// NeuroPLC — Auto-generated IEC 61131-3 SCL
// Graph: mlp | Target: S71500Backend
// Work memory: 1500KB | LUT points: 50
// Nodes: 8 | Ops: {'matmul': 4, 'standard_act': 2, 'softmax': 1, 'argmax': 1}


DATA_BLOCK "NeuroPLC_Weights"
{ S7_Optimized_Access := 'TRUE' }
VERSION : 0.1
NON_RETAIN

   // MatMul 'fc0': W(32×28) + b(32)
   w0 : Array[0..927] of Real :=
    -0.3770078, 0.3990264, 0.0025516, -0.3593162, 0.1366495, -0.1900285, 0.3891852, -0.1283031,
    -0.3550550, 0.1385999, -0.1855089, -0.3235317, 0.0377216, 0.0437886, -0.2197258, 0.2710523,
    0.4527306, -0.1735796, 0.0918002, -0.2219930, -0.0682289, 0.3726985, -0.4032513, 0.3372299,
    0.1742865, 0.2319893, -0.2549221, -0.3851188, -0.3359332, -0.2109050, 0.2084537, -0.2210156,
    0.2307264, -0.0688108, -0.2107350, -0.1310564, 0.3618010, -0.4616588, 0.1129379, -0.1005827,
    0.2574511, 0.3509765, -0.4043934, 0.0268684, 0.2414633, -0.3012495, -0.1214860, 0.1826331,
    0.1323289, -0.0577001, -0.2709421, -0.1641499, 0.2732217, 0.2441040, -0.0308854, 0.3765655,
    0.4575288, 0.1005922, 0.3384550, 0.3164120, -0.0432535, 0.3674217, 0.2929774, 0.2869964,
    0.4056299, 0.2586457, 0.2159618, -0.0111895, 0.2763612, 0.0318691, -0.2383231, -0.2375112,
    0.1950580, 0.2183585, 0.1430424, 0.1642818, 0.4228715, 0.0093872, -0.1228594, 0.2401115,
    0.3953689, -0.1619427, -0.2964523, 0.2409901, 0.0609418, 0.3946368, 0.4126152, -0.3121379,
    -0.3586196, -0.1127610, 0.1867079, 0.3760083, 0.1564328, 0.1040223, 0.0017305, 0.2251267,
    0.0116038, -0.2901824, -0.0485687, -0.0362714, 0.3139654, 0.1739885, 0.0861147, 0.1815197,
    0.4443266, 0.0452933, 0.2375669, 0.3032796, -0.0065490, 0.0947488, 0.1205690, -0.0489962,
    0.1248455, 0.1040717, -0.1340234, -0.1683266, 0.3904992, 0.0068606, 0.1146591, 0.1519284,
    -0.1746107, -0.2354044, 0.1875906, -0.4197009, -0.4406405, 0.4352002, -0.0388191, -0.0047498,
    -0.1199415, 0.2349747, -0.1049938, -0.1901883, 0.2878532, 0.4529921, 0.1495441, -0.1968838,
    -0.0352187, 0.4251530, 0.1424237, -0.0494499, -0.4578539, 0.4085145, -0.1283757, -0.0146367,
    -0.2926642, -0.3105487, 0.4060314, 0.0523238, -0.0729639, -0.3611083, -0.0152973, -0.2996246,
    -0.1483008, -0.2005807, 0.1901999, 0.2505888, -0.0889782, 0.1222107, 0.2931683, -0.1687088,
    0.3804313, -0.2401819, -0.4427654, -0.1597484, -0.0234017, 0.4053880, 0.1999425, 0.0897930,
    0.2230566, -0.3996429, 0.3089489, -0.1815336, 0.2569048, 0.1170700, 0.4507902, -0.2491009,
    -0.2851968, -0.2911826, 0.1435003, 0.0769116, 0.4312512, 0.1906601, 0.1582011, 0.1911615,
    0.1755516, 0.2151861, 0.1524143, -0.3416874, 0.0968710, 0.2657734, 0.4344491, -0.0455045,
    -0.1944677, 0.0802603, -0.1177095, -0.4598294, -0.3312993, 0.0755498, -0.0593091, 0.0803323,
    0.1532357, 0.2834364, -0.2322901, 0.4257076, 0.0440407, 0.4518892, 0.4534211, -0.2465478,
    -0.2583436, 0.1793744, 0.2255728, -0.1181495, 0.0309696, 0.3416602, 0.1074045, -0.3817922,
    0.2319592, 0.2352205, -0.4058878, -0.2966217, -0.4578832, -0.2983192, 0.1998009, -0.3207857,
    0.1968070, 0.0317941, -0.0459040, 0.4509210, -0.4601454, -0.1890926, -0.3331718, 0.3348714,
    -0.1590407, 0.3725954, -0.3415731, 0.2348770, 0.1108938, -0.1082903, 0.2208081, -0.1398732,
    -0.3844526, -0.3700836, -0.1193436, -0.2816384, 0.2890902, -0.0631509, 0.3378636, -0.3628213,
    0.2885490, 0.4045010, 0.0093051, -0.2111615, 0.3647634, -0.3044274, 0.1587412, -0.1364376,
    0.1600578, -0.1415112, 0.3835287, 0.3839180, 0.3733947, -0.4293965, 0.0489564, 0.3753224,
    -0.4217085, 0.3634868, -0.2955091, -0.0699292, -0.2384017, -0.0102885, -0.3535956, -0.0170217,
    0.1624044, -0.4275157, -0.1322644, -0.2605817, -0.3170779, 0.1670513, 0.4262077, -0.2839059,
    -0.0945041, 0.3597159, -0.3709145, -0.0047849, 0.2313926, -0.1789500, 0.1915937, -0.0686558,
    -0.2433297, 0.2847788, -0.1959274, 0.4444867, -0.3373163, 0.3626398, 0.2917026, 0.2028044,
    0.4221848, -0.4179994, -0.3500787, 0.0961545, -0.2199030, 0.0822042, -0.2083196, 0.0249158,
    -0.4572761, -0.1632026, 0.1749700, -0.0869716, -0.1697042, 0.3751226, 0.1738271, 0.4329614,
    -0.1956948, 0.3490632, -0.3649426, -0.0563313, -0.0793010, -0.4472082, -0.1367153, -0.3672275,
    -0.1686790, 0.1854602, -0.0619579, -0.2322961, 0.1377802, -0.2005911, -0.4102385, 0.1393445,
    0.3889906, -0.1450376, 0.2812740, -0.4401638, -0.3213005, 0.4492195, -0.1869051, 0.2014702,
    0.2808036, 0.0341860, -0.1947227, -0.3475538, -0.0703401, -0.1828323, 0.1945061, 0.2123439,
    0.0289259, -0.4163403, 0.3227376, 0.3735557, 0.4516948, 0.0354091, 0.0885729, 0.3177436,
    -0.0816920, 0.4074438, 0.0901380, -0.2812819, -0.0550214, -0.2856297, 0.0293392, 0.2980039,
    0.4104808, 0.4249691, 0.1168610, 0.0088301, 0.0894373, 0.0541764, -0.3080776, -0.2124508,
    -0.4531886, -0.2822830, 0.4012364, 0.1393107, -0.4608335, -0.3710103, -0.1662148, -0.2561499,
    -0.2994817, -0.3900864, -0.1527744, -0.2041700, 0.4141680, -0.1684453, 0.3008100, -0.0788763,
    -0.1708886, 0.4370478, -0.3517387, -0.2863962, 0.1372241, 0.3990270, -0.0800875, -0.4599121,
    -0.3576341, -0.0551274, -0.1279431, -0.3195898, -0.2090862, 0.3166915, -0.4374981, -0.1036189,
    0.2476588, 0.4534730, 0.0433177, -0.1513664, -0.4313229, 0.3424428, -0.3700289, 0.2864294,
    0.3598893, 0.3942130, 0.4272956, -0.1312214, 0.4043608, -0.1855474, 0.4244733, 0.0673699,
    0.3097988, 0.0743738, -0.0575414, -0.0659323, 0.2604717, 0.2774075, 0.1212956, 0.1247821,
    -0.2054413, -0.4303877, 0.2234309, 0.2691470, 0.2036369, 0.2406268, 0.0806441, -0.0397540,
    0.3085780, 0.3872851, 0.4342453, 0.4615774, -0.0954479, -0.3792063, 0.0337596, 0.1248933,
    -0.3579498, -0.4301034, -0.3439160, 0.2736909, 0.2820499, 0.2041379, 0.3628798, -0.0164372,
    0.4257082, 0.1716245, -0.1405404, -0.1675903, -0.0966237, 0.4509315, -0.2013150, 0.1879556,
    -0.1654160, -0.0369867, -0.1594908, 0.3557843, -0.3484282, 0.0975260, 0.2554502, -0.4486252,
    0.1693635, -0.4568610, -0.0845270, 0.1362543, 0.1075566, -0.4298026, -0.2078513, 0.1131138,
    0.4552583, 0.0955319, -0.0176407, 0.2070304, 0.3496518, 0.0070432, 0.3477424, -0.3328675,
    -0.1949137, -0.4457208, 0.1203264, 0.2554769, -0.4579822, 0.1879786, -0.1129094, 0.2853004,
    0.0644755, -0.3809112, -0.1140574, 0.4154554, 0.1054994, 0.4068863, -0.2891253, 0.0136368,
    -0.0689342, -0.4286978, 0.2200271, 0.0348938, -0.3910995, 0.4048684, -0.4127417, -0.2598001,
    0.2112517, -0.1751920, -0.4369283, -0.1871661, 0.0023222, 0.4015321, 0.2616409, -0.3857000,
    -0.2690184, 0.3857079, -0.2387726, 0.2434377, 0.0714437, 0.0578954, -0.2566555, 0.2605321,
    0.0101752, 0.1413683, 0.0509943, -0.3524976, 0.1041765, 0.4223077, 0.3136883, 0.1300556,
    0.4291077, 0.2816193, 0.1022774, -0.3548588, 0.0421972, -0.2862138, -0.0118091, -0.4334079,
    -0.1866055, 0.0868014, 0.1372423, -0.1925206, 0.0754342, -0.1125624, 0.4365539, 0.2470605,
    0.4543210, -0.2610196, 0.2990730, -0.3651120, 0.1277550, 0.2837237, -0.0998289, 0.0588385,
    0.3020812, 0.3680393, -0.3858286, 0.0961783, 0.4596364, -0.2120740, -0.4344158, -0.3728840,
    0.1881307, -0.1419628, -0.2620887, -0.1069769, 0.1167762, 0.0211368, 0.1347501, -0.3661770,
    0.0150048, -0.3614159, 0.2448329, 0.2522876, 0.1993004, -0.0491755, -0.3745691, -0.2868368,
    -0.3422473, 0.2306486, -0.0107990, -0.2471329, 0.4094761, 0.4462330, -0.1006898, -0.3417571,
    -0.3526864, 0.3459129, -0.1873048, -0.3418673, 0.1899261, -0.4220347, 0.4099078, -0.0792820,
    0.4320456, -0.1785485, 0.3833564, -0.1475922, 0.2927010, -0.3002279, 0.4024807, -0.2212537,
    0.1185881, 0.0967595, -0.2608397, -0.0318049, -0.0925073, -0.0683086, -0.4334753, -0.3877276,
    0.2818044, 0.3985909, 0.1276854, 0.1431718, 0.0759905, 0.2359956, -0.3075322, -0.4488399,
    0.3382713, 0.0587753, 0.1603718, 0.2061060, 0.4003389, 0.0745798, -0.1383399, 0.0690251,
    -0.3627133, -0.2600157, 0.2113945, -0.0398504, 0.3121908, -0.0397190, -0.2176074, 0.2885886,
    0.2448370, 0.2249159, 0.3732608, 0.1413454, 0.2938702, 0.0381091, -0.0704973, -0.0676246,
    -0.3967757, 0.1924810, 0.0945449, -0.2569663, 0.0901330, -0.1480842, -0.1106209, -0.0419426,
    0.1201892, -0.3996566, 0.1597114, 0.1156000, -0.3738315, -0.0122839, 0.0922182, 0.1364632,
    -0.0856640, 0.3560283, 0.4043280, -0.2908444, 0.1349952, -0.4130700, -0.4436539, -0.1325469,
    -0.1949083, -0.0976171, 0.1365751, -0.2287472, 0.2230470, -0.2904527, -0.1090742, 0.2397174,
    0.2679743, 0.4155956, 0.4056778, -0.2658896, -0.2220807, -0.4523228, 0.0380185, 0.2802896,
    -0.3090282, -0.0251335, 0.2784542, -0.1911104, 0.1081119, -0.1071131, -0.2883627, 0.1024943,
    0.1079664, 0.0528435, 0.0637380, 0.1360845, 0.2319627, -0.4568143, 0.1126708, 0.2881851,
    -0.0390266, -0.3154065, -0.1891240, 0.3152807, -0.3991016, -0.1147000, -0.1755120, -0.0517076,
    0.2942899, -0.1193079, 0.3693818, 0.3813385, -0.3667921, 0.3955849, -0.3730764, 0.2449901,
    0.4367092, -0.4306898, -0.0932055, -0.2762457, 0.0764579, -0.0612213, 0.3295913, 0.1819134,
    0.3777595, -0.2319842, -0.2136903, -0.0318793, -0.3945642, 0.4148945, 0.1171657, 0.1796898,
    -0.3446222, -0.2104773, 0.0936033, -0.2603089, -0.2805420, -0.4435062, 0.3793530, 0.0610302,
    0.2015716, -0.3638270, 0.0155152, -0.2831283, -0.4584919, 0.3411648, -0.0253624, 0.0896016,
    -0.3085061, 0.3751078, 0.3812718, -0.2918622, 0.2093002, -0.3870984, -0.4346099, 0.3052061,
    0.2963735, -0.4020928, -0.1916119, 0.4596418, -0.2036503, -0.1675266, -0.3643405, -0.0234888,
    0.1632566, 0.2617638, -0.0987748, 0.2144748, 0.3578448, 0.4327554, -0.2301966, -0.1355437,
    0.3251480, -0.0650652, 0.4607093, 0.4538801, 0.3257216, 0.2937019, 0.2583465, 0.0784602,
    -0.2065715, 0.2250659, 0.4356502, -0.0072217, -0.1376927, 0.0364345, -0.3187408, 0.3734230,
    -0.2510726, -0.1775467, -0.3211187, -0.3278403, -0.3991595, 0.0120480, 0.4284748, 0.1523868,
    0.2492753, -0.4192764, -0.4125061, -0.1992944, -0.3151319, -0.4228379, 0.2395529, -0.3589366,
    -0.4471393, 0.1070668, 0.0736012, -0.1881842, 0.1677683, -0.2855140, 0.0012233, -0.4301678,
    0.4539815, -0.2786066, -0.4277930, 0.1925392, -0.4242253, 0.0287630, 0.3206151, 0.4489035,
    -0.3228373, 0.0110811, 0.1304550, 0.3193927, -0.1024946, -0.3389935, -0.0040539, -0.3283602,
    0.3610852, 0.3990757, 0.3903281, 0.2358855, 0.3887415, -0.4240198, 0.1866908, -0.4352202,
    0.4117475, -0.3510597, -0.3075358, -0.4001069, -0.3420205, 0.3339028, -0.1180067, -0.0772094,
    0.2149267, -0.3405320, -0.2175644, 0.2114443, -0.0852025, -0.1429342, -0.4322555, -0.0152842,
    -0.3777024, 0.3303320, 0.0268890, 0.0038649, 0.2427567, -0.1545651, -0.0877347, 0.1801398,
    -0.0444975, 0.2461711, -0.4585460, -0.4603382, 0.3602494, -0.3180314, 0.4038997, 0.3527558,
    0.0713230, -0.0322537, -0.0798554, -0.3169685, 0.2551405, -0.1615019, 0.1647311, 0.4458464,
    0.2310456, -0.0397924, -0.0218926, -0.2396226, -0.2713118, -0.1628663, 0.1717695, 0.1115326,
    -0.1871466, -0.2292732, 0.0375844, 0.2459664, 0.4030566, -0.3787265, 0.2261490, 0.2506774,
    0.0796954, -0.3811616, -0.4266883, -0.4610847, -0.2181492, 0.0805867, -0.1990638, -0.3294418,
    0.0, 0.0, 0.0, 0.0, 0.0, 0.0, 0.0, 0.0,
    0.0, 0.0, 0.0, 0.0, 0.0, 0.0, 0.0, 0.0,
    0.0, 0.0, 0.0, 0.0, 0.0, 0.0, 0.0, 0.0,
    0.0, 0.0, 0.0, 0.0, 0.0, 0.0, 0.0, 0.0;

   // MatMul 'fc1': W(16×32) + b(16)
   w1 : Array[0..527] of Real :=
    -0.3935522, -0.1891568, -0.2444881, -0.2520988, 0.0168740, -0.0661420, -0.0739836, 0.1249234,
    0.0495841, -0.3324362, 0.3990199, -0.3827971, 0.1509344, 0.2727351, 0.1899064, 0.1232548,
    -0.1740977, 0.3996815, -0.0156190, 0.4319531, 0.2304519, 0.2019619, -0.1108288, 0.2639450,
    -0.3004889, 0.2053759, -0.2507130, -0.1099108, 0.3508554, 0.2798605, 0.3080718, -0.2521698,
    0.0398361, 0.0467716, 0.3878656, -0.0975975, 0.2259126, -0.2130022, 0.2817706, -0.4208167,
    0.2917084, 0.4064464, 0.1718341, 0.1449949, -0.2451592, 0.2201938, -0.1602577, -0.3822802,
    -0.1150226, -0.2497750, -0.4201412, -0.0156258, -0.1511233, -0.3021594, -0.1100701, 0.3851436,
    -0.2900417, 0.1651725, 0.2725570, -0.2857571, -0.1159424, 0.3958912, -0.4076339, 0.2155754,
    -0.3153985, 0.1522842, 0.2238676, 0.0359937, -0.2988871, -0.1637969, 0.2320338, 0.0857368,
    0.1976208, 0.0608633, -0.1173251, -0.3213641, -0.0849160, 0.1718496, 0.1879434, 0.3173548,
    0.1776288, -0.2859888, 0.4273638, -0.0753660, 0.2396645, -0.1966574, 0.3941564, -0.4111311,
    0.4031409, 0.3382389, 0.2827366, 0.3812202, -0.4018011, 0.2268997, -0.4327545, 0.0562466,
    -0.4181275, 0.0895361, 0.0215759, -0.4292598, -0.0456185, 0.3361736, 0.1588783, -0.3002315,
    0.1648912, 0.2550659, 0.1932670, 0.3281942, 0.2067506, -0.4133190, -0.1431655, 0.4150747,
    0.3473578, 0.3837779, 0.0933603, 0.2324348, 0.2446682, -0.2923857, -0.1816045, 0.0872757,
    -0.1632624, 0.0132405, 0.0319080, -0.3656984, -0.0171522, 0.4021245, -0.4298175, -0.1553442,
    -0.0378739, -0.0558841, -0.1237145, 0.2343058, -0.3540494, 0.0363749, -0.1224368, 0.1096888,
    0.1723547, 0.2546408, 0.3474467, -0.2087996, 0.4150974, 0.2533172, -0.3616572, -0.1398576,
    0.1326821, 0.0146453, 0.3335588, 0.1515740, -0.1683524, -0.0804338, 0.4306846, 0.0640880,
    0.2288128, 0.0326079, 0.1973397, 0.0868359, 0.3189215, 0.1261115, 0.4030693, 0.0196063,
    0.1143374, -0.1861071, -0.3970583, 0.4306547, 0.3728819, -0.1188974, -0.2829262, -0.3271297,
    -0.2453017, 0.1782900, -0.0166697, -0.3631355, -0.1097839, 0.0609611, 0.0001612, 0.3813087,
    0.1942296, -0.3436415, -0.3196552, -0.3243870, 0.2198140, 0.3918344, 0.0912264, 0.2238992,
    -0.3022591, 0.3621037, 0.3434459, -0.1731028, 0.3113935, 0.3348374, 0.2629885, 0.0019000,
    0.3024160, -0.0626668, -0.0818046, -0.3892852, -0.1082816, -0.2291101, 0.1406163, -0.3290255,
    0.0634920, -0.0686606, 0.1352782, -0.2557390, 0.3506733, -0.2629621, -0.2691220, -0.2397180,
    -0.2910091, 0.0893200, 0.1797454, 0.2301134, -0.3933525, 0.0697611, -0.1224633, -0.1336698,
    0.0822801, 0.0491940, 0.1768592, -0.1431975, 0.1519364, 0.2522070, -0.3521394, -0.3634867,
    0.3611591, 0.0925913, 0.3470873, 0.0306298, 0.3107211, -0.1883461, 0.2165535, -0.1091567,
    0.0689959, 0.3486420, -0.1837859, 0.0694401, 0.2055986, 0.2386295, 0.3321949, 0.1919344,
    0.4253771, -0.3774826, -0.0617012, 0.0334252, 0.3778329, 0.2201037, -0.2276398, 0.1301410,
    0.3501653, 0.2798014, 0.4256953, -0.1441793, -0.0663480, -0.4205136, 0.3892752, -0.3286948,
    0.0955538, 0.3663456, -0.1591998, 0.3128131, 0.0344288, 0.0733947, -0.2083270, -0.3181835,
    0.2916943, 0.1976334, -0.0215316, -0.1335652, -0.1110399, -0.4227563, -0.2664171, 0.4199895,
    -0.3832088, 0.0912991, 0.3962664, -0.2253252, -0.4168374, -0.0803243, -0.2418978, 0.2176948,
    -0.3986563, -0.0865313, -0.1186279, -0.4000811, 0.0561389, -0.1613197, -0.4163839, 0.1215905,
    -0.1568890, 0.3878794, 0.3653413, -0.2158771, -0.0794441, 0.0936781, 0.2255915, 0.3624552,
    0.2718166, -0.0088999, -0.2009125, 0.0077918, 0.1461028, 0.2432971, 0.1760126, 0.1427329,
    -0.0146298, -0.3526535, -0.1145816, 0.0303672, -0.3133373, 0.3928600, 0.3592887, 0.3393191,
    0.2999697, -0.2127717, -0.3682398, -0.2014481, 0.2898328, -0.0393004, 0.3296660, -0.2576033,
    -0.2580386, 0.3286115, 0.3484521, 0.1741413, -0.3222574, 0.4139940, -0.2123599, -0.0532465,
    -0.1246679, -0.1157071, -0.3183327, 0.0137842, 0.1334311, -0.0707376, -0.1285511, -0.4081723,
    -0.1506712, 0.2322767, 0.0759037, 0.3221440, 0.2789797, -0.3218980, -0.0615748, -0.3991559,
    -0.4185835, -0.2636460, -0.1289205, 0.2750368, 0.2876762, -0.3447819, -0.1141558, 0.1948618,
    -0.1709883, 0.3542524, -0.1556085, -0.0569944, 0.2803813, 0.0518793, -0.0245967, 0.1485651,
    -0.0932260, 0.2044456, -0.3843631, 0.1491727, -0.1015462, 0.0335794, -0.2548426, -0.2155586,
    0.3438183, -0.3987876, -0.1833805, -0.3147031, -0.4217897, 0.4175099, -0.0144855, -0.3033746,
    -0.1601701, 0.3044005, -0.0549371, -0.2065555, -0.2234019, -0.3457984, -0.0095058, 0.4049891,
    0.1624429, -0.0648286, 0.3860819, 0.1274094, 0.2339818, 0.1994726, -0.3863117, -0.3547160,
    0.2731713, 0.3852477, -0.0738010, 0.4109565, 0.3464701, 0.2911135, -0.2596304, -0.3724965,
    -0.0749315, -0.0193869, -0.2211102, -0.2740593, -0.3613006, 0.2223929, -0.0702648, 0.1260325,
    -0.3447631, 0.2582121, 0.1769404, 0.4101386, -0.2221670, 0.4048361, -0.2569288, 0.1401117,
    -0.3058916, 0.2899141, -0.2516046, -0.0204311, 0.3705838, 0.4224865, -0.0464628, 0.2932765,
    -0.1048749, -0.1260871, 0.1966383, 0.3772893, 0.0665107, 0.4117973, 0.3348016, -0.3298126,
    0.1286661, -0.3882708, 0.0985853, 0.2120279, 0.2686936, -0.2604558, -0.1903019, 0.1670984,
    0.1759086, -0.2155941, -0.4271439, -0.1347190, 0.3518137, 0.1066233, -0.0060884, -0.0989732,
    -0.1571809, 0.2292162, -0.2883213, 0.1154139, 0.2343982, -0.0461321, -0.2751803, -0.0112296,
    0.2915563, 0.3558245, 0.2112975, -0.2306676, -0.3320167, 0.2315517, -0.0035513, 0.3149335,
    0.0999751, -0.0704947, -0.3919639, -0.0087440, -0.1189045, -0.3321721, 0.0222524, -0.3617505,
    -0.1745312, 0.0928437, 0.3209649, 0.4192130, 0.0815147, 0.2839914, 0.0094900, 0.3304590,
    0.1507888, -0.1633613, -0.2137657, 0.4228123, -0.0633699, -0.3235189, -0.3633914, 0.0783406,
    0.2527627, 0.4272875, -0.2854069, 0.1855697, -0.1320681, 0.3007466, 0.0956593, -0.2299400,
    0.0410553, 0.0255588, -0.2430910, 0.1599361, 0.2384051, 0.0154256, 0.2833597, 0.0843526,
    0.3284023, 0.1945453, 0.1661874, 0.1049307, -0.3034132, 0.1947828, 0.3134930, -0.1473352,
    0.0, 0.0, 0.0, 0.0, 0.0, 0.0, 0.0, 0.0,
    0.0, 0.0, 0.0, 0.0, 0.0, 0.0, 0.0, 0.0;

   // MatMul 'fc2': W(4×16) + b(4)
   w2 : Array[0..67] of Real :=
    0.3119249, -0.6119898, 0.2570214, -0.5775461, -0.3303460, -0.0226893, -0.0253589, 0.0133041,
    0.2119226, 0.1795658, 0.1164464, -0.5784835, 0.4102349, -0.5724207, -0.5247188, 0.2892720,
    0.0710802, 0.4088987, -0.4011595, 0.1927266, 0.0227786, -0.3939466, 0.5633335, 0.4811944,
    0.4671021, -0.4038831, 0.2076768, -0.5081061, 0.1620483, -0.2713509, 0.4681324, 0.3022301,
    0.3770372, -0.5370517, -0.1928490, 0.0872999, -0.0823838, -0.2322832, 0.0953737, -0.0633100,
    -0.2465645, 0.4775037, 0.5268021, -0.1162953, -0.3230001, 0.2317193, 0.2054757, -0.4918106,
    0.2500432, -0.1568022, -0.4481698, 0.3745956, -0.0458250, -0.5208440, 0.1315344, 0.3012816,
    0.4046838, -0.6074986, 0.0947582, -0.3567927, 0.0561409, 0.1993957, 0.1098667, 0.0024996,
    0.0, 0.0, 0.0, 0.0;

   // Total: 3 array blocks
END_DATA_BLOCK

FUNCTION_BLOCK "NeuroPLC_Inference"
{ S7_Optimized_Access := 'TRUE' }
VERSION : 0.1
VAR_INPUT
    features : Array[0..27] of Real;
END_VAR

VAR_OUTPUT
    fault_class : Int;
    confidence : Real;
END_VAR

VAR
    i, j, k : Int;
    sum_val, max_val, t_val : Real;
    v0 : Array[0..27] of Real;
    v1 : Array[0..31] of Real;
    v2 : Array[0..31] of Real;
    v3 : Array[0..15] of Real;
    v4 : Array[0..15] of Real;
    v5 : Array[0..3] of Real;
    v6 : Array[0..3] of Real;
END_VAR

BEGIN
    // ---- Input ----
    FOR i := 0 TO 27 DO
        v0[i] := features[i];
    END_FOR;

    // ---- fc0: MatMul(28→32) ----
    // W = "NeuroPLC_Weights".w0[:896],   b = w0[896:]
    v1[0] := "NeuroPLC_Weights".w0[896 + 0] + "NeuroPLC_Weights".w0[0] * v0[0] + "NeuroPLC_Weights".w0[1] * v0[1] + "NeuroPLC_Weights".w0[2] * v0[2] + "NeuroPLC_Weights".w0[3] * v0[3] + "NeuroPLC_Weights".w0[4] * v0[4] + "NeuroPLC_Weights".w0[5] * v0[5] + "NeuroPLC_Weights".w0[6] * v0[6] + "NeuroPLC_Weights".w0[7] * v0[7] + "NeuroPLC_Weights".w0[8] * v0[8] + "NeuroPLC_Weights".w0[9] * v0[9] + "NeuroPLC_Weights".w0[10] * v0[10] + "NeuroPLC_Weights".w0[11] * v0[11] + "NeuroPLC_Weights".w0[12] * v0[12] + "NeuroPLC_Weights".w0[13] * v0[13] + "NeuroPLC_Weights".w0[14] * v0[14] + "NeuroPLC_Weights".w0[15] * v0[15] + "NeuroPLC_Weights".w0[16] * v0[16] + "NeuroPLC_Weights".w0[17] * v0[17] + "NeuroPLC_Weights".w0[18] * v0[18] + "NeuroPLC_Weights".w0[19] * v0[19] + "NeuroPLC_Weights".w0[20] * v0[20] + "NeuroPLC_Weights".w0[21] * v0[21] + "NeuroPLC_Weights".w0[22] * v0[22] + "NeuroPLC_Weights".w0[23] * v0[23] + "NeuroPLC_Weights".w0[24] * v0[24] + "NeuroPLC_Weights".w0[25] * v0[25] + "NeuroPLC_Weights".w0[26] * v0[26] + "NeuroPLC_Weights".w0[27] * v0[27];
    v1[1] := "NeuroPLC_Weights".w0[896 + 1] + "NeuroPLC_Weights".w0[28] * v0[0] + "NeuroPLC_Weights".w0[29] * v0[1] + "NeuroPLC_Weights".w0[30] * v0[2] + "NeuroPLC_Weights".w0[31] * v0[3] + "NeuroPLC_Weights".w0[32] * v0[4] + "NeuroPLC_Weights".w0[33] * v0[5] + "NeuroPLC_Weights".w0[34] * v0[6] + "NeuroPLC_Weights".w0[35] * v0[7] + "NeuroPLC_Weights".w0[36] * v0[8] + "NeuroPLC_Weights".w0[37] * v0[9] + "NeuroPLC_Weights".w0[38] * v0[10] + "NeuroPLC_Weights".w0[39] * v0[11] + "NeuroPLC_Weights".w0[40] * v0[12] + "NeuroPLC_Weights".w0[41] * v0[13] + "NeuroPLC_Weights".w0[42] * v0[14] + "NeuroPLC_Weights".w0[43] * v0[15] + "NeuroPLC_Weights".w0[44] * v0[16] + "NeuroPLC_Weights".w0[45] * v0[17] + "NeuroPLC_Weights".w0[46] * v0[18] + "NeuroPLC_Weights".w0[47] * v0[19] + "NeuroPLC_Weights".w0[48] * v0[20] + "NeuroPLC_Weights".w0[49] * v0[21] + "NeuroPLC_Weights".w0[50] * v0[22] + "NeuroPLC_Weights".w0[51] * v0[23] + "NeuroPLC_Weights".w0[52] * v0[24] + "NeuroPLC_Weights".w0[53] * v0[25] + "NeuroPLC_Weights".w0[54] * v0[26] + "NeuroPLC_Weights".w0[55] * v0[27];
    v1[2] := "NeuroPLC_Weights".w0[896 + 2] + "NeuroPLC_Weights".w0[56] * v0[0] + "NeuroPLC_Weights".w0[57] * v0[1] + "NeuroPLC_Weights".w0[58] * v0[2] + "NeuroPLC_Weights".w0[59] * v0[3] + "NeuroPLC_Weights".w0[60] * v0[4] + "NeuroPLC_Weights".w0[61] * v0[5] + "NeuroPLC_Weights".w0[62] * v0[6] + "NeuroPLC_Weights".w0[63] * v0[7] + "NeuroPLC_Weights".w0[64] * v0[8] + "NeuroPLC_Weights".w0[65] * v0[9] + "NeuroPLC_Weights".w0[66] * v0[10] + "NeuroPLC_Weights".w0[67] * v0[11] + "NeuroPLC_Weights".w0[68] * v0[12] + "NeuroPLC_Weights".w0[69] * v0[13] + "NeuroPLC_Weights".w0[70] * v0[14] + "NeuroPLC_Weights".w0[71] * v0[15] + "NeuroPLC_Weights".w0[72] * v0[16] + "NeuroPLC_Weights".w0[73] * v0[17] + "NeuroPLC_Weights".w0[74] * v0[18] + "NeuroPLC_Weights".w0[75] * v0[19] + "NeuroPLC_Weights".w0[76] * v0[20] + "NeuroPLC_Weights".w0[77] * v0[21] + "NeuroPLC_Weights".w0[78] * v0[22] + "NeuroPLC_Weights".w0[79] * v0[23] + "NeuroPLC_Weights".w0[80] * v0[24] + "NeuroPLC_Weights".w0[81] * v0[25] + "NeuroPLC_Weights".w0[82] * v0[26] + "NeuroPLC_Weights".w0[83] * v0[27];
    v1[3] := "NeuroPLC_Weights".w0[896 + 3] + "NeuroPLC_Weights".w0[84] * v0[0] + "NeuroPLC_Weights".w0[85] * v0[1] + "NeuroPLC_Weights".w0[86] * v0[2] + "NeuroPLC_Weights".w0[87] * v0[3] + "NeuroPLC_Weights".w0[88] * v0[4] + "NeuroPLC_Weights".w0[89] * v0[5] + "NeuroPLC_Weights".w0[90] * v0[6] + "NeuroPLC_Weights".w0[91] * v0[7] + "NeuroPLC_Weights".w0[92] * v0[8] + "NeuroPLC_Weights".w0[93] * v0[9] + "NeuroPLC_Weights".w0[94] * v0[10] + "NeuroPLC_Weights".w0[95] * v0[11] + "NeuroPLC_Weights".w0[96] * v0[12] + "NeuroPLC_Weights".w0[97] * v0[13] + "NeuroPLC_Weights".w0[98] * v0[14] + "NeuroPLC_Weights".w0[99] * v0[15] + "NeuroPLC_Weights".w0[100] * v0[16] + "NeuroPLC_Weights".w0[101] * v0[17] + "NeuroPLC_Weights".w0[102] * v0[18] + "NeuroPLC_Weights".w0[103] * v0[19] + "NeuroPLC_Weights".w0[104] * v0[20] + "NeuroPLC_Weights".w0[105] * v0[21] + "NeuroPLC_Weights".w0[106] * v0[22] + "NeuroPLC_Weights".w0[107] * v0[23] + "NeuroPLC_Weights".w0[108] * v0[24] + "NeuroPLC_Weights".w0[109] * v0[25] + "NeuroPLC_Weights".w0[110] * v0[26] + "NeuroPLC_Weights".w0[111] * v0[27];
    v1[4] := "NeuroPLC_Weights".w0[896 + 4] + "NeuroPLC_Weights".w0[112] * v0[0] + "NeuroPLC_Weights".w0[113] * v0[1] + "NeuroPLC_Weights".w0[114] * v0[2] + "NeuroPLC_Weights".w0[115] * v0[3] + "NeuroPLC_Weights".w0[116] * v0[4] + "NeuroPLC_Weights".w0[117] * v0[5] + "NeuroPLC_Weights".w0[118] * v0[6] + "NeuroPLC_Weights".w0[119] * v0[7] + "NeuroPLC_Weights".w0[120] * v0[8] + "NeuroPLC_Weights".w0[121] * v0[9] + "NeuroPLC_Weights".w0[122] * v0[10] + "NeuroPLC_Weights".w0[123] * v0[11] + "NeuroPLC_Weights".w0[124] * v0[12] + "NeuroPLC_Weights".w0[125] * v0[13] + "NeuroPLC_Weights".w0[126] * v0[14] + "NeuroPLC_Weights".w0[127] * v0[15] + "NeuroPLC_Weights".w0[128] * v0[16] + "NeuroPLC_Weights".w0[129] * v0[17] + "NeuroPLC_Weights".w0[130] * v0[18] + "NeuroPLC_Weights".w0[131] * v0[19] + "NeuroPLC_Weights".w0[132] * v0[20] + "NeuroPLC_Weights".w0[133] * v0[21] + "NeuroPLC_Weights".w0[134] * v0[22] + "NeuroPLC_Weights".w0[135] * v0[23] + "NeuroPLC_Weights".w0[136] * v0[24] + "NeuroPLC_Weights".w0[137] * v0[25] + "NeuroPLC_Weights".w0[138] * v0[26] + "NeuroPLC_Weights".w0[139] * v0[27];
    v1[5] := "NeuroPLC_Weights".w0[896 + 5] + "NeuroPLC_Weights".w0[140] * v0[0] + "NeuroPLC_Weights".w0[141] * v0[1] + "NeuroPLC_Weights".w0[142] * v0[2] + "NeuroPLC_Weights".w0[143] * v0[3] + "NeuroPLC_Weights".w0[144] * v0[4] + "NeuroPLC_Weights".w0[145] * v0[5] + "NeuroPLC_Weights".w0[146] * v0[6] + "NeuroPLC_Weights".w0[147] * v0[7] + "NeuroPLC_Weights".w0[148] * v0[8] + "NeuroPLC_Weights".w0[149] * v0[9] + "NeuroPLC_Weights".w0[150] * v0[10] + "NeuroPLC_Weights".w0[151] * v0[11] + "NeuroPLC_Weights".w0[152] * v0[12] + "NeuroPLC_Weights".w0[153] * v0[13] + "NeuroPLC_Weights".w0[154] * v0[14] + "NeuroPLC_Weights".w0[155] * v0[15] + "NeuroPLC_Weights".w0[156] * v0[16] + "NeuroPLC_Weights".w0[157] * v0[17] + "NeuroPLC_Weights".w0[158] * v0[18] + "NeuroPLC_Weights".w0[159] * v0[19] + "NeuroPLC_Weights".w0[160] * v0[20] + "NeuroPLC_Weights".w0[161] * v0[21] + "NeuroPLC_Weights".w0[162] * v0[22] + "NeuroPLC_Weights".w0[163] * v0[23] + "NeuroPLC_Weights".w0[164] * v0[24] + "NeuroPLC_Weights".w0[165] * v0[25] + "NeuroPLC_Weights".w0[166] * v0[26] + "NeuroPLC_Weights".w0[167] * v0[27];
    v1[6] := "NeuroPLC_Weights".w0[896 + 6] + "NeuroPLC_Weights".w0[168] * v0[0] + "NeuroPLC_Weights".w0[169] * v0[1] + "NeuroPLC_Weights".w0[170] * v0[2] + "NeuroPLC_Weights".w0[171] * v0[3] + "NeuroPLC_Weights".w0[172] * v0[4] + "NeuroPLC_Weights".w0[173] * v0[5] + "NeuroPLC_Weights".w0[174] * v0[6] + "NeuroPLC_Weights".w0[175] * v0[7] + "NeuroPLC_Weights".w0[176] * v0[8] + "NeuroPLC_Weights".w0[177] * v0[9] + "NeuroPLC_Weights".w0[178] * v0[10] + "NeuroPLC_Weights".w0[179] * v0[11] + "NeuroPLC_Weights".w0[180] * v0[12] + "NeuroPLC_Weights".w0[181] * v0[13] + "NeuroPLC_Weights".w0[182] * v0[14] + "NeuroPLC_Weights".w0[183] * v0[15] + "NeuroPLC_Weights".w0[184] * v0[16] + "NeuroPLC_Weights".w0[185] * v0[17] + "NeuroPLC_Weights".w0[186] * v0[18] + "NeuroPLC_Weights".w0[187] * v0[19] + "NeuroPLC_Weights".w0[188] * v0[20] + "NeuroPLC_Weights".w0[189] * v0[21] + "NeuroPLC_Weights".w0[190] * v0[22] + "NeuroPLC_Weights".w0[191] * v0[23] + "NeuroPLC_Weights".w0[192] * v0[24] + "NeuroPLC_Weights".w0[193] * v0[25] + "NeuroPLC_Weights".w0[194] * v0[26] + "NeuroPLC_Weights".w0[195] * v0[27];
    v1[7] := "NeuroPLC_Weights".w0[896 + 7] + "NeuroPLC_Weights".w0[196] * v0[0] + "NeuroPLC_Weights".w0[197] * v0[1] + "NeuroPLC_Weights".w0[198] * v0[2] + "NeuroPLC_Weights".w0[199] * v0[3] + "NeuroPLC_Weights".w0[200] * v0[4] + "NeuroPLC_Weights".w0[201] * v0[5] + "NeuroPLC_Weights".w0[202] * v0[6] + "NeuroPLC_Weights".w0[203] * v0[7] + "NeuroPLC_Weights".w0[204] * v0[8] + "NeuroPLC_Weights".w0[205] * v0[9] + "NeuroPLC_Weights".w0[206] * v0[10] + "NeuroPLC_Weights".w0[207] * v0[11] + "NeuroPLC_Weights".w0[208] * v0[12] + "NeuroPLC_Weights".w0[209] * v0[13] + "NeuroPLC_Weights".w0[210] * v0[14] + "NeuroPLC_Weights".w0[211] * v0[15] + "NeuroPLC_Weights".w0[212] * v0[16] + "NeuroPLC_Weights".w0[213] * v0[17] + "NeuroPLC_Weights".w0[214] * v0[18] + "NeuroPLC_Weights".w0[215] * v0[19] + "NeuroPLC_Weights".w0[216] * v0[20] + "NeuroPLC_Weights".w0[217] * v0[21] + "NeuroPLC_Weights".w0[218] * v0[22] + "NeuroPLC_Weights".w0[219] * v0[23] + "NeuroPLC_Weights".w0[220] * v0[24] + "NeuroPLC_Weights".w0[221] * v0[25] + "NeuroPLC_Weights".w0[222] * v0[26] + "NeuroPLC_Weights".w0[223] * v0[27];
    v1[8] := "NeuroPLC_Weights".w0[896 + 8] + "NeuroPLC_Weights".w0[224] * v0[0] + "NeuroPLC_Weights".w0[225] * v0[1] + "NeuroPLC_Weights".w0[226] * v0[2] + "NeuroPLC_Weights".w0[227] * v0[3] + "NeuroPLC_Weights".w0[228] * v0[4] + "NeuroPLC_Weights".w0[229] * v0[5] + "NeuroPLC_Weights".w0[230] * v0[6] + "NeuroPLC_Weights".w0[231] * v0[7] + "NeuroPLC_Weights".w0[232] * v0[8] + "NeuroPLC_Weights".w0[233] * v0[9] + "NeuroPLC_Weights".w0[234] * v0[10] + "NeuroPLC_Weights".w0[235] * v0[11] + "NeuroPLC_Weights".w0[236] * v0[12] + "NeuroPLC_Weights".w0[237] * v0[13] + "NeuroPLC_Weights".w0[238] * v0[14] + "NeuroPLC_Weights".w0[239] * v0[15] + "NeuroPLC_Weights".w0[240] * v0[16] + "NeuroPLC_Weights".w0[241] * v0[17] + "NeuroPLC_Weights".w0[242] * v0[18] + "NeuroPLC_Weights".w0[243] * v0[19] + "NeuroPLC_Weights".w0[244] * v0[20] + "NeuroPLC_Weights".w0[245] * v0[21] + "NeuroPLC_Weights".w0[246] * v0[22] + "NeuroPLC_Weights".w0[247] * v0[23] + "NeuroPLC_Weights".w0[248] * v0[24] + "NeuroPLC_Weights".w0[249] * v0[25] + "NeuroPLC_Weights".w0[250] * v0[26] + "NeuroPLC_Weights".w0[251] * v0[27];
    v1[9] := "NeuroPLC_Weights".w0[896 + 9] + "NeuroPLC_Weights".w0[252] * v0[0] + "NeuroPLC_Weights".w0[253] * v0[1] + "NeuroPLC_Weights".w0[254] * v0[2] + "NeuroPLC_Weights".w0[255] * v0[3] + "NeuroPLC_Weights".w0[256] * v0[4] + "NeuroPLC_Weights".w0[257] * v0[5] + "NeuroPLC_Weights".w0[258] * v0[6] + "NeuroPLC_Weights".w0[259] * v0[7] + "NeuroPLC_Weights".w0[260] * v0[8] + "NeuroPLC_Weights".w0[261] * v0[9] + "NeuroPLC_Weights".w0[262] * v0[10] + "NeuroPLC_Weights".w0[263] * v0[11] + "NeuroPLC_Weights".w0[264] * v0[12] + "NeuroPLC_Weights".w0[265] * v0[13] + "NeuroPLC_Weights".w0[266] * v0[14] + "NeuroPLC_Weights".w0[267] * v0[15] + "NeuroPLC_Weights".w0[268] * v0[16] + "NeuroPLC_Weights".w0[269] * v0[17] + "NeuroPLC_Weights".w0[270] * v0[18] + "NeuroPLC_Weights".w0[271] * v0[19] + "NeuroPLC_Weights".w0[272] * v0[20] + "NeuroPLC_Weights".w0[273] * v0[21] + "NeuroPLC_Weights".w0[274] * v0[22] + "NeuroPLC_Weights".w0[275] * v0[23] + "NeuroPLC_Weights".w0[276] * v0[24] + "NeuroPLC_Weights".w0[277] * v0[25] + "NeuroPLC_Weights".w0[278] * v0[26] + "NeuroPLC_Weights".w0[279] * v0[27];
    v1[10] := "NeuroPLC_Weights".w0[896 + 10] + "NeuroPLC_Weights".w0[280] * v0[0] + "NeuroPLC_Weights".w0[281] * v0[1] + "NeuroPLC_Weights".w0[282] * v0[2] + "NeuroPLC_Weights".w0[283] * v0[3] + "NeuroPLC_Weights".w0[284] * v0[4] + "NeuroPLC_Weights".w0[285] * v0[5] + "NeuroPLC_Weights".w0[286] * v0[6] + "NeuroPLC_Weights".w0[287] * v0[7] + "NeuroPLC_Weights".w0[288] * v0[8] + "NeuroPLC_Weights".w0[289] * v0[9] + "NeuroPLC_Weights".w0[290] * v0[10] + "NeuroPLC_Weights".w0[291] * v0[11] + "NeuroPLC_Weights".w0[292] * v0[12] + "NeuroPLC_Weights".w0[293] * v0[13] + "NeuroPLC_Weights".w0[294] * v0[14] + "NeuroPLC_Weights".w0[295] * v0[15] + "NeuroPLC_Weights".w0[296] * v0[16] + "NeuroPLC_Weights".w0[297] * v0[17] + "NeuroPLC_Weights".w0[298] * v0[18] + "NeuroPLC_Weights".w0[299] * v0[19] + "NeuroPLC_Weights".w0[300] * v0[20] + "NeuroPLC_Weights".w0[301] * v0[21] + "NeuroPLC_Weights".w0[302] * v0[22] + "NeuroPLC_Weights".w0[303] * v0[23] + "NeuroPLC_Weights".w0[304] * v0[24] + "NeuroPLC_Weights".w0[305] * v0[25] + "NeuroPLC_Weights".w0[306] * v0[26] + "NeuroPLC_Weights".w0[307] * v0[27];
    v1[11] := "NeuroPLC_Weights".w0[896 + 11] + "NeuroPLC_Weights".w0[308] * v0[0] + "NeuroPLC_Weights".w0[309] * v0[1] + "NeuroPLC_Weights".w0[310] * v0[2] + "NeuroPLC_Weights".w0[311] * v0[3] + "NeuroPLC_Weights".w0[312] * v0[4] + "NeuroPLC_Weights".w0[313] * v0[5] + "NeuroPLC_Weights".w0[314] * v0[6] + "NeuroPLC_Weights".w0[315] * v0[7] + "NeuroPLC_Weights".w0[316] * v0[8] + "NeuroPLC_Weights".w0[317] * v0[9] + "NeuroPLC_Weights".w0[318] * v0[10] + "NeuroPLC_Weights".w0[319] * v0[11] + "NeuroPLC_Weights".w0[320] * v0[12] + "NeuroPLC_Weights".w0[321] * v0[13] + "NeuroPLC_Weights".w0[322] * v0[14] + "NeuroPLC_Weights".w0[323] * v0[15] + "NeuroPLC_Weights".w0[324] * v0[16] + "NeuroPLC_Weights".w0[325] * v0[17] + "NeuroPLC_Weights".w0[326] * v0[18] + "NeuroPLC_Weights".w0[327] * v0[19] + "NeuroPLC_Weights".w0[328] * v0[20] + "NeuroPLC_Weights".w0[329] * v0[21] + "NeuroPLC_Weights".w0[330] * v0[22] + "NeuroPLC_Weights".w0[331] * v0[23] + "NeuroPLC_Weights".w0[332] * v0[24] + "NeuroPLC_Weights".w0[333] * v0[25] + "NeuroPLC_Weights".w0[334] * v0[26] + "NeuroPLC_Weights".w0[335] * v0[27];
    v1[12] := "NeuroPLC_Weights".w0[896 + 12] + "NeuroPLC_Weights".w0[336] * v0[0] + "NeuroPLC_Weights".w0[337] * v0[1] + "NeuroPLC_Weights".w0[338] * v0[2] + "NeuroPLC_Weights".w0[339] * v0[3] + "NeuroPLC_Weights".w0[340] * v0[4] + "NeuroPLC_Weights".w0[341] * v0[5] + "NeuroPLC_Weights".w0[342] * v0[6] + "NeuroPLC_Weights".w0[343] * v0[7] + "NeuroPLC_Weights".w0[344] * v0[8] + "NeuroPLC_Weights".w0[345] * v0[9] + "NeuroPLC_Weights".w0[346] * v0[10] + "NeuroPLC_Weights".w0[347] * v0[11] + "NeuroPLC_Weights".w0[348] * v0[12] + "NeuroPLC_Weights".w0[349] * v0[13] + "NeuroPLC_Weights".w0[350] * v0[14] + "NeuroPLC_Weights".w0[351] * v0[15] + "NeuroPLC_Weights".w0[352] * v0[16] + "NeuroPLC_Weights".w0[353] * v0[17] + "NeuroPLC_Weights".w0[354] * v0[18] + "NeuroPLC_Weights".w0[355] * v0[19] + "NeuroPLC_Weights".w0[356] * v0[20] + "NeuroPLC_Weights".w0[357] * v0[21] + "NeuroPLC_Weights".w0[358] * v0[22] + "NeuroPLC_Weights".w0[359] * v0[23] + "NeuroPLC_Weights".w0[360] * v0[24] + "NeuroPLC_Weights".w0[361] * v0[25] + "NeuroPLC_Weights".w0[362] * v0[26] + "NeuroPLC_Weights".w0[363] * v0[27];
    v1[13] := "NeuroPLC_Weights".w0[896 + 13] + "NeuroPLC_Weights".w0[364] * v0[0] + "NeuroPLC_Weights".w0[365] * v0[1] + "NeuroPLC_Weights".w0[366] * v0[2] + "NeuroPLC_Weights".w0[367] * v0[3] + "NeuroPLC_Weights".w0[368] * v0[4] + "NeuroPLC_Weights".w0[369] * v0[5] + "NeuroPLC_Weights".w0[370] * v0[6] + "NeuroPLC_Weights".w0[371] * v0[7] + "NeuroPLC_Weights".w0[372] * v0[8] + "NeuroPLC_Weights".w0[373] * v0[9] + "NeuroPLC_Weights".w0[374] * v0[10] + "NeuroPLC_Weights".w0[375] * v0[11] + "NeuroPLC_Weights".w0[376] * v0[12] + "NeuroPLC_Weights".w0[377] * v0[13] + "NeuroPLC_Weights".w0[378] * v0[14] + "NeuroPLC_Weights".w0[379] * v0[15] + "NeuroPLC_Weights".w0[380] * v0[16] + "NeuroPLC_Weights".w0[381] * v0[17] + "NeuroPLC_Weights".w0[382] * v0[18] + "NeuroPLC_Weights".w0[383] * v0[19] + "NeuroPLC_Weights".w0[384] * v0[20] + "NeuroPLC_Weights".w0[385] * v0[21] + "NeuroPLC_Weights".w0[386] * v0[22] + "NeuroPLC_Weights".w0[387] * v0[23] + "NeuroPLC_Weights".w0[388] * v0[24] + "NeuroPLC_Weights".w0[389] * v0[25] + "NeuroPLC_Weights".w0[390] * v0[26] + "NeuroPLC_Weights".w0[391] * v0[27];
    v1[14] := "NeuroPLC_Weights".w0[896 + 14] + "NeuroPLC_Weights".w0[392] * v0[0] + "NeuroPLC_Weights".w0[393] * v0[1] + "NeuroPLC_Weights".w0[394] * v0[2] + "NeuroPLC_Weights".w0[395] * v0[3] + "NeuroPLC_Weights".w0[396] * v0[4] + "NeuroPLC_Weights".w0[397] * v0[5] + "NeuroPLC_Weights".w0[398] * v0[6] + "NeuroPLC_Weights".w0[399] * v0[7] + "NeuroPLC_Weights".w0[400] * v0[8] + "NeuroPLC_Weights".w0[401] * v0[9] + "NeuroPLC_Weights".w0[402] * v0[10] + "NeuroPLC_Weights".w0[403] * v0[11] + "NeuroPLC_Weights".w0[404] * v0[12] + "NeuroPLC_Weights".w0[405] * v0[13] + "NeuroPLC_Weights".w0[406] * v0[14] + "NeuroPLC_Weights".w0[407] * v0[15] + "NeuroPLC_Weights".w0[408] * v0[16] + "NeuroPLC_Weights".w0[409] * v0[17] + "NeuroPLC_Weights".w0[410] * v0[18] + "NeuroPLC_Weights".w0[411] * v0[19] + "NeuroPLC_Weights".w0[412] * v0[20] + "NeuroPLC_Weights".w0[413] * v0[21] + "NeuroPLC_Weights".w0[414] * v0[22] + "NeuroPLC_Weights".w0[415] * v0[23] + "NeuroPLC_Weights".w0[416] * v0[24] + "NeuroPLC_Weights".w0[417] * v0[25] + "NeuroPLC_Weights".w0[418] * v0[26] + "NeuroPLC_Weights".w0[419] * v0[27];
    v1[15] := "NeuroPLC_Weights".w0[896 + 15] + "NeuroPLC_Weights".w0[420] * v0[0] + "NeuroPLC_Weights".w0[421] * v0[1] + "NeuroPLC_Weights".w0[422] * v0[2] + "NeuroPLC_Weights".w0[423] * v0[3] + "NeuroPLC_Weights".w0[424] * v0[4] + "NeuroPLC_Weights".w0[425] * v0[5] + "NeuroPLC_Weights".w0[426] * v0[6] + "NeuroPLC_Weights".w0[427] * v0[7] + "NeuroPLC_Weights".w0[428] * v0[8] + "NeuroPLC_Weights".w0[429] * v0[9] + "NeuroPLC_Weights".w0[430] * v0[10] + "NeuroPLC_Weights".w0[431] * v0[11] + "NeuroPLC_Weights".w0[432] * v0[12] + "NeuroPLC_Weights".w0[433] * v0[13] + "NeuroPLC_Weights".w0[434] * v0[14] + "NeuroPLC_Weights".w0[435] * v0[15] + "NeuroPLC_Weights".w0[436] * v0[16] + "NeuroPLC_Weights".w0[437] * v0[17] + "NeuroPLC_Weights".w0[438] * v0[18] + "NeuroPLC_Weights".w0[439] * v0[19] + "NeuroPLC_Weights".w0[440] * v0[20] + "NeuroPLC_Weights".w0[441] * v0[21] + "NeuroPLC_Weights".w0[442] * v0[22] + "NeuroPLC_Weights".w0[443] * v0[23] + "NeuroPLC_Weights".w0[444] * v0[24] + "NeuroPLC_Weights".w0[445] * v0[25] + "NeuroPLC_Weights".w0[446] * v0[26] + "NeuroPLC_Weights".w0[447] * v0[27];
    v1[16] := "NeuroPLC_Weights".w0[896 + 16] + "NeuroPLC_Weights".w0[448] * v0[0] + "NeuroPLC_Weights".w0[449] * v0[1] + "NeuroPLC_Weights".w0[450] * v0[2] + "NeuroPLC_Weights".w0[451] * v0[3] + "NeuroPLC_Weights".w0[452] * v0[4] + "NeuroPLC_Weights".w0[453] * v0[5] + "NeuroPLC_Weights".w0[454] * v0[6] + "NeuroPLC_Weights".w0[455] * v0[7] + "NeuroPLC_Weights".w0[456] * v0[8] + "NeuroPLC_Weights".w0[457] * v0[9] + "NeuroPLC_Weights".w0[458] * v0[10] + "NeuroPLC_Weights".w0[459] * v0[11] + "NeuroPLC_Weights".w0[460] * v0[12] + "NeuroPLC_Weights".w0[461] * v0[13] + "NeuroPLC_Weights".w0[462] * v0[14] + "NeuroPLC_Weights".w0[463] * v0[15] + "NeuroPLC_Weights".w0[464] * v0[16] + "NeuroPLC_Weights".w0[465] * v0[17] + "NeuroPLC_Weights".w0[466] * v0[18] + "NeuroPLC_Weights".w0[467] * v0[19] + "NeuroPLC_Weights".w0[468] * v0[20] + "NeuroPLC_Weights".w0[469] * v0[21] + "NeuroPLC_Weights".w0[470] * v0[22] + "NeuroPLC_Weights".w0[471] * v0[23] + "NeuroPLC_Weights".w0[472] * v0[24] + "NeuroPLC_Weights".w0[473] * v0[25] + "NeuroPLC_Weights".w0[474] * v0[26] + "NeuroPLC_Weights".w0[475] * v0[27];
    v1[17] := "NeuroPLC_Weights".w0[896 + 17] + "NeuroPLC_Weights".w0[476] * v0[0] + "NeuroPLC_Weights".w0[477] * v0[1] + "NeuroPLC_Weights".w0[478] * v0[2] + "NeuroPLC_Weights".w0[479] * v0[3] + "NeuroPLC_Weights".w0[480] * v0[4] + "NeuroPLC_Weights".w0[481] * v0[5] + "NeuroPLC_Weights".w0[482] * v0[6] + "NeuroPLC_Weights".w0[483] * v0[7] + "NeuroPLC_Weights".w0[484] * v0[8] + "NeuroPLC_Weights".w0[485] * v0[9] + "NeuroPLC_Weights".w0[486] * v0[10] + "NeuroPLC_Weights".w0[487] * v0[11] + "NeuroPLC_Weights".w0[488] * v0[12] + "NeuroPLC_Weights".w0[489] * v0[13] + "NeuroPLC_Weights".w0[490] * v0[14] + "NeuroPLC_Weights".w0[491] * v0[15] + "NeuroPLC_Weights".w0[492] * v0[16] + "NeuroPLC_Weights".w0[493] * v0[17] + "NeuroPLC_Weights".w0[494] * v0[18] + "NeuroPLC_Weights".w0[495] * v0[19] + "NeuroPLC_Weights".w0[496] * v0[20] + "NeuroPLC_Weights".w0[497] * v0[21] + "NeuroPLC_Weights".w0[498] * v0[22] + "NeuroPLC_Weights".w0[499] * v0[23] + "NeuroPLC_Weights".w0[500] * v0[24] + "NeuroPLC_Weights".w0[501] * v0[25] + "NeuroPLC_Weights".w0[502] * v0[26] + "NeuroPLC_Weights".w0[503] * v0[27];
    v1[18] := "NeuroPLC_Weights".w0[896 + 18] + "NeuroPLC_Weights".w0[504] * v0[0] + "NeuroPLC_Weights".w0[505] * v0[1] + "NeuroPLC_Weights".w0[506] * v0[2] + "NeuroPLC_Weights".w0[507] * v0[3] + "NeuroPLC_Weights".w0[508] * v0[4] + "NeuroPLC_Weights".w0[509] * v0[5] + "NeuroPLC_Weights".w0[510] * v0[6] + "NeuroPLC_Weights".w0[511] * v0[7] + "NeuroPLC_Weights".w0[512] * v0[8] + "NeuroPLC_Weights".w0[513] * v0[9] + "NeuroPLC_Weights".w0[514] * v0[10] + "NeuroPLC_Weights".w0[515] * v0[11] + "NeuroPLC_Weights".w0[516] * v0[12] + "NeuroPLC_Weights".w0[517] * v0[13] + "NeuroPLC_Weights".w0[518] * v0[14] + "NeuroPLC_Weights".w0[519] * v0[15] + "NeuroPLC_Weights".w0[520] * v0[16] + "NeuroPLC_Weights".w0[521] * v0[17] + "NeuroPLC_Weights".w0[522] * v0[18] + "NeuroPLC_Weights".w0[523] * v0[19] + "NeuroPLC_Weights".w0[524] * v0[20] + "NeuroPLC_Weights".w0[525] * v0[21] + "NeuroPLC_Weights".w0[526] * v0[22] + "NeuroPLC_Weights".w0[527] * v0[23] + "NeuroPLC_Weights".w0[528] * v0[24] + "NeuroPLC_Weights".w0[529] * v0[25] + "NeuroPLC_Weights".w0[530] * v0[26] + "NeuroPLC_Weights".w0[531] * v0[27];
    v1[19] := "NeuroPLC_Weights".w0[896 + 19] + "NeuroPLC_Weights".w0[532] * v0[0] + "NeuroPLC_Weights".w0[533] * v0[1] + "NeuroPLC_Weights".w0[534] * v0[2] + "NeuroPLC_Weights".w0[535] * v0[3] + "NeuroPLC_Weights".w0[536] * v0[4] + "NeuroPLC_Weights".w0[537] * v0[5] + "NeuroPLC_Weights".w0[538] * v0[6] + "NeuroPLC_Weights".w0[539] * v0[7] + "NeuroPLC_Weights".w0[540] * v0[8] + "NeuroPLC_Weights".w0[541] * v0[9] + "NeuroPLC_Weights".w0[542] * v0[10] + "NeuroPLC_Weights".w0[543] * v0[11] + "NeuroPLC_Weights".w0[544] * v0[12] + "NeuroPLC_Weights".w0[545] * v0[13] + "NeuroPLC_Weights".w0[546] * v0[14] + "NeuroPLC_Weights".w0[547] * v0[15] + "NeuroPLC_Weights".w0[548] * v0[16] + "NeuroPLC_Weights".w0[549] * v0[17] + "NeuroPLC_Weights".w0[550] * v0[18] + "NeuroPLC_Weights".w0[551] * v0[19] + "NeuroPLC_Weights".w0[552] * v0[20] + "NeuroPLC_Weights".w0[553] * v0[21] + "NeuroPLC_Weights".w0[554] * v0[22] + "NeuroPLC_Weights".w0[555] * v0[23] + "NeuroPLC_Weights".w0[556] * v0[24] + "NeuroPLC_Weights".w0[557] * v0[25] + "NeuroPLC_Weights".w0[558] * v0[26] + "NeuroPLC_Weights".w0[559] * v0[27];
    v1[20] := "NeuroPLC_Weights".w0[896 + 20] + "NeuroPLC_Weights".w0[560] * v0[0] + "NeuroPLC_Weights".w0[561] * v0[1] + "NeuroPLC_Weights".w0[562] * v0[2] + "NeuroPLC_Weights".w0[563] * v0[3] + "NeuroPLC_Weights".w0[564] * v0[4] + "NeuroPLC_Weights".w0[565] * v0[5] + "NeuroPLC_Weights".w0[566] * v0[6] + "NeuroPLC_Weights".w0[567] * v0[7] + "NeuroPLC_Weights".w0[568] * v0[8] + "NeuroPLC_Weights".w0[569] * v0[9] + "NeuroPLC_Weights".w0[570] * v0[10] + "NeuroPLC_Weights".w0[571] * v0[11] + "NeuroPLC_Weights".w0[572] * v0[12] + "NeuroPLC_Weights".w0[573] * v0[13] + "NeuroPLC_Weights".w0[574] * v0[14] + "NeuroPLC_Weights".w0[575] * v0[15] + "NeuroPLC_Weights".w0[576] * v0[16] + "NeuroPLC_Weights".w0[577] * v0[17] + "NeuroPLC_Weights".w0[578] * v0[18] + "NeuroPLC_Weights".w0[579] * v0[19] + "NeuroPLC_Weights".w0[580] * v0[20] + "NeuroPLC_Weights".w0[581] * v0[21] + "NeuroPLC_Weights".w0[582] * v0[22] + "NeuroPLC_Weights".w0[583] * v0[23] + "NeuroPLC_Weights".w0[584] * v0[24] + "NeuroPLC_Weights".w0[585] * v0[25] + "NeuroPLC_Weights".w0[586] * v0[26] + "NeuroPLC_Weights".w0[587] * v0[27];
    v1[21] := "NeuroPLC_Weights".w0[896 + 21] + "NeuroPLC_Weights".w0[588] * v0[0] + "NeuroPLC_Weights".w0[589] * v0[1] + "NeuroPLC_Weights".w0[590] * v0[2] + "NeuroPLC_Weights".w0[591] * v0[3] + "NeuroPLC_Weights".w0[592] * v0[4] + "NeuroPLC_Weights".w0[593] * v0[5] + "NeuroPLC_Weights".w0[594] * v0[6] + "NeuroPLC_Weights".w0[595] * v0[7] + "NeuroPLC_Weights".w0[596] * v0[8] + "NeuroPLC_Weights".w0[597] * v0[9] + "NeuroPLC_Weights".w0[598] * v0[10] + "NeuroPLC_Weights".w0[599] * v0[11] + "NeuroPLC_Weights".w0[600] * v0[12] + "NeuroPLC_Weights".w0[601] * v0[13] + "NeuroPLC_Weights".w0[602] * v0[14] + "NeuroPLC_Weights".w0[603] * v0[15] + "NeuroPLC_Weights".w0[604] * v0[16] + "NeuroPLC_Weights".w0[605] * v0[17] + "NeuroPLC_Weights".w0[606] * v0[18] + "NeuroPLC_Weights".w0[607] * v0[19] + "NeuroPLC_Weights".w0[608] * v0[20] + "NeuroPLC_Weights".w0[609] * v0[21] + "NeuroPLC_Weights".w0[610] * v0[22] + "NeuroPLC_Weights".w0[611] * v0[23] + "NeuroPLC_Weights".w0[612] * v0[24] + "NeuroPLC_Weights".w0[613] * v0[25] + "NeuroPLC_Weights".w0[614] * v0[26] + "NeuroPLC_Weights".w0[615] * v0[27];
    v1[22] := "NeuroPLC_Weights".w0[896 + 22] + "NeuroPLC_Weights".w0[616] * v0[0] + "NeuroPLC_Weights".w0[617] * v0[1] + "NeuroPLC_Weights".w0[618] * v0[2] + "NeuroPLC_Weights".w0[619] * v0[3] + "NeuroPLC_Weights".w0[620] * v0[4] + "NeuroPLC_Weights".w0[621] * v0[5] + "NeuroPLC_Weights".w0[622] * v0[6] + "NeuroPLC_Weights".w0[623] * v0[7] + "NeuroPLC_Weights".w0[624] * v0[8] + "NeuroPLC_Weights".w0[625] * v0[9] + "NeuroPLC_Weights".w0[626] * v0[10] + "NeuroPLC_Weights".w0[627] * v0[11] + "NeuroPLC_Weights".w0[628] * v0[12] + "NeuroPLC_Weights".w0[629] * v0[13] + "NeuroPLC_Weights".w0[630] * v0[14] + "NeuroPLC_Weights".w0[631] * v0[15] + "NeuroPLC_Weights".w0[632] * v0[16] + "NeuroPLC_Weights".w0[633] * v0[17] + "NeuroPLC_Weights".w0[634] * v0[18] + "NeuroPLC_Weights".w0[635] * v0[19] + "NeuroPLC_Weights".w0[636] * v0[20] + "NeuroPLC_Weights".w0[637] * v0[21] + "NeuroPLC_Weights".w0[638] * v0[22] + "NeuroPLC_Weights".w0[639] * v0[23] + "NeuroPLC_Weights".w0[640] * v0[24] + "NeuroPLC_Weights".w0[641] * v0[25] + "NeuroPLC_Weights".w0[642] * v0[26] + "NeuroPLC_Weights".w0[643] * v0[27];
    v1[23] := "NeuroPLC_Weights".w0[896 + 23] + "NeuroPLC_Weights".w0[644] * v0[0] + "NeuroPLC_Weights".w0[645] * v0[1] + "NeuroPLC_Weights".w0[646] * v0[2] + "NeuroPLC_Weights".w0[647] * v0[3] + "NeuroPLC_Weights".w0[648] * v0[4] + "NeuroPLC_Weights".w0[649] * v0[5] + "NeuroPLC_Weights".w0[650] * v0[6] + "NeuroPLC_Weights".w0[651] * v0[7] + "NeuroPLC_Weights".w0[652] * v0[8] + "NeuroPLC_Weights".w0[653] * v0[9] + "NeuroPLC_Weights".w0[654] * v0[10] + "NeuroPLC_Weights".w0[655] * v0[11] + "NeuroPLC_Weights".w0[656] * v0[12] + "NeuroPLC_Weights".w0[657] * v0[13] + "NeuroPLC_Weights".w0[658] * v0[14] + "NeuroPLC_Weights".w0[659] * v0[15] + "NeuroPLC_Weights".w0[660] * v0[16] + "NeuroPLC_Weights".w0[661] * v0[17] + "NeuroPLC_Weights".w0[662] * v0[18] + "NeuroPLC_Weights".w0[663] * v0[19] + "NeuroPLC_Weights".w0[664] * v0[20] + "NeuroPLC_Weights".w0[665] * v0[21] + "NeuroPLC_Weights".w0[666] * v0[22] + "NeuroPLC_Weights".w0[667] * v0[23] + "NeuroPLC_Weights".w0[668] * v0[24] + "NeuroPLC_Weights".w0[669] * v0[25] + "NeuroPLC_Weights".w0[670] * v0[26] + "NeuroPLC_Weights".w0[671] * v0[27];
    v1[24] := "NeuroPLC_Weights".w0[896 + 24] + "NeuroPLC_Weights".w0[672] * v0[0] + "NeuroPLC_Weights".w0[673] * v0[1] + "NeuroPLC_Weights".w0[674] * v0[2] + "NeuroPLC_Weights".w0[675] * v0[3] + "NeuroPLC_Weights".w0[676] * v0[4] + "NeuroPLC_Weights".w0[677] * v0[5] + "NeuroPLC_Weights".w0[678] * v0[6] + "NeuroPLC_Weights".w0[679] * v0[7] + "NeuroPLC_Weights".w0[680] * v0[8] + "NeuroPLC_Weights".w0[681] * v0[9] + "NeuroPLC_Weights".w0[682] * v0[10] + "NeuroPLC_Weights".w0[683] * v0[11] + "NeuroPLC_Weights".w0[684] * v0[12] + "NeuroPLC_Weights".w0[685] * v0[13] + "NeuroPLC_Weights".w0[686] * v0[14] + "NeuroPLC_Weights".w0[687] * v0[15] + "NeuroPLC_Weights".w0[688] * v0[16] + "NeuroPLC_Weights".w0[689] * v0[17] + "NeuroPLC_Weights".w0[690] * v0[18] + "NeuroPLC_Weights".w0[691] * v0[19] + "NeuroPLC_Weights".w0[692] * v0[20] + "NeuroPLC_Weights".w0[693] * v0[21] + "NeuroPLC_Weights".w0[694] * v0[22] + "NeuroPLC_Weights".w0[695] * v0[23] + "NeuroPLC_Weights".w0[696] * v0[24] + "NeuroPLC_Weights".w0[697] * v0[25] + "NeuroPLC_Weights".w0[698] * v0[26] + "NeuroPLC_Weights".w0[699] * v0[27];
    v1[25] := "NeuroPLC_Weights".w0[896 + 25] + "NeuroPLC_Weights".w0[700] * v0[0] + "NeuroPLC_Weights".w0[701] * v0[1] + "NeuroPLC_Weights".w0[702] * v0[2] + "NeuroPLC_Weights".w0[703] * v0[3] + "NeuroPLC_Weights".w0[704] * v0[4] + "NeuroPLC_Weights".w0[705] * v0[5] + "NeuroPLC_Weights".w0[706] * v0[6] + "NeuroPLC_Weights".w0[707] * v0[7] + "NeuroPLC_Weights".w0[708] * v0[8] + "NeuroPLC_Weights".w0[709] * v0[9] + "NeuroPLC_Weights".w0[710] * v0[10] + "NeuroPLC_Weights".w0[711] * v0[11] + "NeuroPLC_Weights".w0[712] * v0[12] + "NeuroPLC_Weights".w0[713] * v0[13] + "NeuroPLC_Weights".w0[714] * v0[14] + "NeuroPLC_Weights".w0[715] * v0[15] + "NeuroPLC_Weights".w0[716] * v0[16] + "NeuroPLC_Weights".w0[717] * v0[17] + "NeuroPLC_Weights".w0[718] * v0[18] + "NeuroPLC_Weights".w0[719] * v0[19] + "NeuroPLC_Weights".w0[720] * v0[20] + "NeuroPLC_Weights".w0[721] * v0[21] + "NeuroPLC_Weights".w0[722] * v0[22] + "NeuroPLC_Weights".w0[723] * v0[23] + "NeuroPLC_Weights".w0[724] * v0[24] + "NeuroPLC_Weights".w0[725] * v0[25] + "NeuroPLC_Weights".w0[726] * v0[26] + "NeuroPLC_Weights".w0[727] * v0[27];
    v1[26] := "NeuroPLC_Weights".w0[896 + 26] + "NeuroPLC_Weights".w0[728] * v0[0] + "NeuroPLC_Weights".w0[729] * v0[1] + "NeuroPLC_Weights".w0[730] * v0[2] + "NeuroPLC_Weights".w0[731] * v0[3] + "NeuroPLC_Weights".w0[732] * v0[4] + "NeuroPLC_Weights".w0[733] * v0[5] + "NeuroPLC_Weights".w0[734] * v0[6] + "NeuroPLC_Weights".w0[735] * v0[7] + "NeuroPLC_Weights".w0[736] * v0[8] + "NeuroPLC_Weights".w0[737] * v0[9] + "NeuroPLC_Weights".w0[738] * v0[10] + "NeuroPLC_Weights".w0[739] * v0[11] + "NeuroPLC_Weights".w0[740] * v0[12] + "NeuroPLC_Weights".w0[741] * v0[13] + "NeuroPLC_Weights".w0[742] * v0[14] + "NeuroPLC_Weights".w0[743] * v0[15] + "NeuroPLC_Weights".w0[744] * v0[16] + "NeuroPLC_Weights".w0[745] * v0[17] + "NeuroPLC_Weights".w0[746] * v0[18] + "NeuroPLC_Weights".w0[747] * v0[19] + "NeuroPLC_Weights".w0[748] * v0[20] + "NeuroPLC_Weights".w0[749] * v0[21] + "NeuroPLC_Weights".w0[750] * v0[22] + "NeuroPLC_Weights".w0[751] * v0[23] + "NeuroPLC_Weights".w0[752] * v0[24] + "NeuroPLC_Weights".w0[753] * v0[25] + "NeuroPLC_Weights".w0[754] * v0[26] + "NeuroPLC_Weights".w0[755] * v0[27];
    v1[27] := "NeuroPLC_Weights".w0[896 + 27] + "NeuroPLC_Weights".w0[756] * v0[0] + "NeuroPLC_Weights".w0[757] * v0[1] + "NeuroPLC_Weights".w0[758] * v0[2] + "NeuroPLC_Weights".w0[759] * v0[3] + "NeuroPLC_Weights".w0[760] * v0[4] + "NeuroPLC_Weights".w0[761] * v0[5] + "NeuroPLC_Weights".w0[762] * v0[6] + "NeuroPLC_Weights".w0[763] * v0[7] + "NeuroPLC_Weights".w0[764] * v0[8] + "NeuroPLC_Weights".w0[765] * v0[9] + "NeuroPLC_Weights".w0[766] * v0[10] + "NeuroPLC_Weights".w0[767] * v0[11] + "NeuroPLC_Weights".w0[768] * v0[12] + "NeuroPLC_Weights".w0[769] * v0[13] + "NeuroPLC_Weights".w0[770] * v0[14] + "NeuroPLC_Weights".w0[771] * v0[15] + "NeuroPLC_Weights".w0[772] * v0[16] + "NeuroPLC_Weights".w0[773] * v0[17] + "NeuroPLC_Weights".w0[774] * v0[18] + "NeuroPLC_Weights".w0[775] * v0[19] + "NeuroPLC_Weights".w0[776] * v0[20] + "NeuroPLC_Weights".w0[777] * v0[21] + "NeuroPLC_Weights".w0[778] * v0[22] + "NeuroPLC_Weights".w0[779] * v0[23] + "NeuroPLC_Weights".w0[780] * v0[24] + "NeuroPLC_Weights".w0[781] * v0[25] + "NeuroPLC_Weights".w0[782] * v0[26] + "NeuroPLC_Weights".w0[783] * v0[27];
    v1[28] := "NeuroPLC_Weights".w0[896 + 28] + "NeuroPLC_Weights".w0[784] * v0[0] + "NeuroPLC_Weights".w0[785] * v0[1] + "NeuroPLC_Weights".w0[786] * v0[2] + "NeuroPLC_Weights".w0[787] * v0[3] + "NeuroPLC_Weights".w0[788] * v0[4] + "NeuroPLC_Weights".w0[789] * v0[5] + "NeuroPLC_Weights".w0[790] * v0[6] + "NeuroPLC_Weights".w0[791] * v0[7] + "NeuroPLC_Weights".w0[792] * v0[8] + "NeuroPLC_Weights".w0[793] * v0[9] + "NeuroPLC_Weights".w0[794] * v0[10] + "NeuroPLC_Weights".w0[795] * v0[11] + "NeuroPLC_Weights".w0[796] * v0[12] + "NeuroPLC_Weights".w0[797] * v0[13] + "NeuroPLC_Weights".w0[798] * v0[14] + "NeuroPLC_Weights".w0[799] * v0[15] + "NeuroPLC_Weights".w0[800] * v0[16] + "NeuroPLC_Weights".w0[801] * v0[17] + "NeuroPLC_Weights".w0[802] * v0[18] + "NeuroPLC_Weights".w0[803] * v0[19] + "NeuroPLC_Weights".w0[804] * v0[20] + "NeuroPLC_Weights".w0[805] * v0[21] + "NeuroPLC_Weights".w0[806] * v0[22] + "NeuroPLC_Weights".w0[807] * v0[23] + "NeuroPLC_Weights".w0[808] * v0[24] + "NeuroPLC_Weights".w0[809] * v0[25] + "NeuroPLC_Weights".w0[810] * v0[26] + "NeuroPLC_Weights".w0[811] * v0[27];
    v1[29] := "NeuroPLC_Weights".w0[896 + 29] + "NeuroPLC_Weights".w0[812] * v0[0] + "NeuroPLC_Weights".w0[813] * v0[1] + "NeuroPLC_Weights".w0[814] * v0[2] + "NeuroPLC_Weights".w0[815] * v0[3] + "NeuroPLC_Weights".w0[816] * v0[4] + "NeuroPLC_Weights".w0[817] * v0[5] + "NeuroPLC_Weights".w0[818] * v0[6] + "NeuroPLC_Weights".w0[819] * v0[7] + "NeuroPLC_Weights".w0[820] * v0[8] + "NeuroPLC_Weights".w0[821] * v0[9] + "NeuroPLC_Weights".w0[822] * v0[10] + "NeuroPLC_Weights".w0[823] * v0[11] + "NeuroPLC_Weights".w0[824] * v0[12] + "NeuroPLC_Weights".w0[825] * v0[13] + "NeuroPLC_Weights".w0[826] * v0[14] + "NeuroPLC_Weights".w0[827] * v0[15] + "NeuroPLC_Weights".w0[828] * v0[16] + "NeuroPLC_Weights".w0[829] * v0[17] + "NeuroPLC_Weights".w0[830] * v0[18] + "NeuroPLC_Weights".w0[831] * v0[19] + "NeuroPLC_Weights".w0[832] * v0[20] + "NeuroPLC_Weights".w0[833] * v0[21] + "NeuroPLC_Weights".w0[834] * v0[22] + "NeuroPLC_Weights".w0[835] * v0[23] + "NeuroPLC_Weights".w0[836] * v0[24] + "NeuroPLC_Weights".w0[837] * v0[25] + "NeuroPLC_Weights".w0[838] * v0[26] + "NeuroPLC_Weights".w0[839] * v0[27];
    v1[30] := "NeuroPLC_Weights".w0[896 + 30] + "NeuroPLC_Weights".w0[840] * v0[0] + "NeuroPLC_Weights".w0[841] * v0[1] + "NeuroPLC_Weights".w0[842] * v0[2] + "NeuroPLC_Weights".w0[843] * v0[3] + "NeuroPLC_Weights".w0[844] * v0[4] + "NeuroPLC_Weights".w0[845] * v0[5] + "NeuroPLC_Weights".w0[846] * v0[6] + "NeuroPLC_Weights".w0[847] * v0[7] + "NeuroPLC_Weights".w0[848] * v0[8] + "NeuroPLC_Weights".w0[849] * v0[9] + "NeuroPLC_Weights".w0[850] * v0[10] + "NeuroPLC_Weights".w0[851] * v0[11] + "NeuroPLC_Weights".w0[852] * v0[12] + "NeuroPLC_Weights".w0[853] * v0[13] + "NeuroPLC_Weights".w0[854] * v0[14] + "NeuroPLC_Weights".w0[855] * v0[15] + "NeuroPLC_Weights".w0[856] * v0[16] + "NeuroPLC_Weights".w0[857] * v0[17] + "NeuroPLC_Weights".w0[858] * v0[18] + "NeuroPLC_Weights".w0[859] * v0[19] + "NeuroPLC_Weights".w0[860] * v0[20] + "NeuroPLC_Weights".w0[861] * v0[21] + "NeuroPLC_Weights".w0[862] * v0[22] + "NeuroPLC_Weights".w0[863] * v0[23] + "NeuroPLC_Weights".w0[864] * v0[24] + "NeuroPLC_Weights".w0[865] * v0[25] + "NeuroPLC_Weights".w0[866] * v0[26] + "NeuroPLC_Weights".w0[867] * v0[27];
    v1[31] := "NeuroPLC_Weights".w0[896 + 31] + "NeuroPLC_Weights".w0[868] * v0[0] + "NeuroPLC_Weights".w0[869] * v0[1] + "NeuroPLC_Weights".w0[870] * v0[2] + "NeuroPLC_Weights".w0[871] * v0[3] + "NeuroPLC_Weights".w0[872] * v0[4] + "NeuroPLC_Weights".w0[873] * v0[5] + "NeuroPLC_Weights".w0[874] * v0[6] + "NeuroPLC_Weights".w0[875] * v0[7] + "NeuroPLC_Weights".w0[876] * v0[8] + "NeuroPLC_Weights".w0[877] * v0[9] + "NeuroPLC_Weights".w0[878] * v0[10] + "NeuroPLC_Weights".w0[879] * v0[11] + "NeuroPLC_Weights".w0[880] * v0[12] + "NeuroPLC_Weights".w0[881] * v0[13] + "NeuroPLC_Weights".w0[882] * v0[14] + "NeuroPLC_Weights".w0[883] * v0[15] + "NeuroPLC_Weights".w0[884] * v0[16] + "NeuroPLC_Weights".w0[885] * v0[17] + "NeuroPLC_Weights".w0[886] * v0[18] + "NeuroPLC_Weights".w0[887] * v0[19] + "NeuroPLC_Weights".w0[888] * v0[20] + "NeuroPLC_Weights".w0[889] * v0[21] + "NeuroPLC_Weights".w0[890] * v0[22] + "NeuroPLC_Weights".w0[891] * v0[23] + "NeuroPLC_Weights".w0[892] * v0[24] + "NeuroPLC_Weights".w0[893] * v0[25] + "NeuroPLC_Weights".w0[894] * v0[26] + "NeuroPLC_Weights".w0[895] * v0[27];

    // ---- relu0: RELU ----
    IF v1[0] > 0.0 THEN v2[0] := v1[0]; ELSE v2[0] := 0.0; END_IF;
    IF v1[1] > 0.0 THEN v2[1] := v1[1]; ELSE v2[1] := 0.0; END_IF;
    IF v1[2] > 0.0 THEN v2[2] := v1[2]; ELSE v2[2] := 0.0; END_IF;
    IF v1[3] > 0.0 THEN v2[3] := v1[3]; ELSE v2[3] := 0.0; END_IF;
    IF v1[4] > 0.0 THEN v2[4] := v1[4]; ELSE v2[4] := 0.0; END_IF;
    IF v1[5] > 0.0 THEN v2[5] := v1[5]; ELSE v2[5] := 0.0; END_IF;
    IF v1[6] > 0.0 THEN v2[6] := v1[6]; ELSE v2[6] := 0.0; END_IF;
    IF v1[7] > 0.0 THEN v2[7] := v1[7]; ELSE v2[7] := 0.0; END_IF;
    IF v1[8] > 0.0 THEN v2[8] := v1[8]; ELSE v2[8] := 0.0; END_IF;
    IF v1[9] > 0.0 THEN v2[9] := v1[9]; ELSE v2[9] := 0.0; END_IF;
    IF v1[10] > 0.0 THEN v2[10] := v1[10]; ELSE v2[10] := 0.0; END_IF;
    IF v1[11] > 0.0 THEN v2[11] := v1[11]; ELSE v2[11] := 0.0; END_IF;
    IF v1[12] > 0.0 THEN v2[12] := v1[12]; ELSE v2[12] := 0.0; END_IF;
    IF v1[13] > 0.0 THEN v2[13] := v1[13]; ELSE v2[13] := 0.0; END_IF;
    IF v1[14] > 0.0 THEN v2[14] := v1[14]; ELSE v2[14] := 0.0; END_IF;
    IF v1[15] > 0.0 THEN v2[15] := v1[15]; ELSE v2[15] := 0.0; END_IF;
    IF v1[16] > 0.0 THEN v2[16] := v1[16]; ELSE v2[16] := 0.0; END_IF;
    IF v1[17] > 0.0 THEN v2[17] := v1[17]; ELSE v2[17] := 0.0; END_IF;
    IF v1[18] > 0.0 THEN v2[18] := v1[18]; ELSE v2[18] := 0.0; END_IF;
    IF v1[19] > 0.0 THEN v2[19] := v1[19]; ELSE v2[19] := 0.0; END_IF;
    IF v1[20] > 0.0 THEN v2[20] := v1[20]; ELSE v2[20] := 0.0; END_IF;
    IF v1[21] > 0.0 THEN v2[21] := v1[21]; ELSE v2[21] := 0.0; END_IF;
    IF v1[22] > 0.0 THEN v2[22] := v1[22]; ELSE v2[22] := 0.0; END_IF;
    IF v1[23] > 0.0 THEN v2[23] := v1[23]; ELSE v2[23] := 0.0; END_IF;
    IF v1[24] > 0.0 THEN v2[24] := v1[24]; ELSE v2[24] := 0.0; END_IF;
    IF v1[25] > 0.0 THEN v2[25] := v1[25]; ELSE v2[25] := 0.0; END_IF;
    IF v1[26] > 0.0 THEN v2[26] := v1[26]; ELSE v2[26] := 0.0; END_IF;
    IF v1[27] > 0.0 THEN v2[27] := v1[27]; ELSE v2[27] := 0.0; END_IF;
    IF v1[28] > 0.0 THEN v2[28] := v1[28]; ELSE v2[28] := 0.0; END_IF;
    IF v1[29] > 0.0 THEN v2[29] := v1[29]; ELSE v2[29] := 0.0; END_IF;
    IF v1[30] > 0.0 THEN v2[30] := v1[30]; ELSE v2[30] := 0.0; END_IF;
    IF v1[31] > 0.0 THEN v2[31] := v1[31]; ELSE v2[31] := 0.0; END_IF;

    // ---- fc1: MatMul(32→16) ----
    // W = "NeuroPLC_Weights".w1[:512],   b = w1[512:]
    v3[0] := "NeuroPLC_Weights".w1[512 + 0] + "NeuroPLC_Weights".w1[0] * v2[0] + "NeuroPLC_Weights".w1[1] * v2[1] + "NeuroPLC_Weights".w1[2] * v2[2] + "NeuroPLC_Weights".w1[3] * v2[3] + "NeuroPLC_Weights".w1[4] * v2[4] + "NeuroPLC_Weights".w1[5] * v2[5] + "NeuroPLC_Weights".w1[6] * v2[6] + "NeuroPLC_Weights".w1[7] * v2[7] + "NeuroPLC_Weights".w1[8] * v2[8] + "NeuroPLC_Weights".w1[9] * v2[9] + "NeuroPLC_Weights".w1[10] * v2[10] + "NeuroPLC_Weights".w1[11] * v2[11] + "NeuroPLC_Weights".w1[12] * v2[12] + "NeuroPLC_Weights".w1[13] * v2[13] + "NeuroPLC_Weights".w1[14] * v2[14] + "NeuroPLC_Weights".w1[15] * v2[15] + "NeuroPLC_Weights".w1[16] * v2[16] + "NeuroPLC_Weights".w1[17] * v2[17] + "NeuroPLC_Weights".w1[18] * v2[18] + "NeuroPLC_Weights".w1[19] * v2[19] + "NeuroPLC_Weights".w1[20] * v2[20] + "NeuroPLC_Weights".w1[21] * v2[21] + "NeuroPLC_Weights".w1[22] * v2[22] + "NeuroPLC_Weights".w1[23] * v2[23] + "NeuroPLC_Weights".w1[24] * v2[24] + "NeuroPLC_Weights".w1[25] * v2[25] + "NeuroPLC_Weights".w1[26] * v2[26] + "NeuroPLC_Weights".w1[27] * v2[27] + "NeuroPLC_Weights".w1[28] * v2[28] + "NeuroPLC_Weights".w1[29] * v2[29] + "NeuroPLC_Weights".w1[30] * v2[30] + "NeuroPLC_Weights".w1[31] * v2[31];
    v3[1] := "NeuroPLC_Weights".w1[512 + 1] + "NeuroPLC_Weights".w1[32] * v2[0] + "NeuroPLC_Weights".w1[33] * v2[1] + "NeuroPLC_Weights".w1[34] * v2[2] + "NeuroPLC_Weights".w1[35] * v2[3] + "NeuroPLC_Weights".w1[36] * v2[4] + "NeuroPLC_Weights".w1[37] * v2[5] + "NeuroPLC_Weights".w1[38] * v2[6] + "NeuroPLC_Weights".w1[39] * v2[7] + "NeuroPLC_Weights".w1[40] * v2[8] + "NeuroPLC_Weights".w1[41] * v2[9] + "NeuroPLC_Weights".w1[42] * v2[10] + "NeuroPLC_Weights".w1[43] * v2[11] + "NeuroPLC_Weights".w1[44] * v2[12] + "NeuroPLC_Weights".w1[45] * v2[13] + "NeuroPLC_Weights".w1[46] * v2[14] + "NeuroPLC_Weights".w1[47] * v2[15] + "NeuroPLC_Weights".w1[48] * v2[16] + "NeuroPLC_Weights".w1[49] * v2[17] + "NeuroPLC_Weights".w1[50] * v2[18] + "NeuroPLC_Weights".w1[51] * v2[19] + "NeuroPLC_Weights".w1[52] * v2[20] + "NeuroPLC_Weights".w1[53] * v2[21] + "NeuroPLC_Weights".w1[54] * v2[22] + "NeuroPLC_Weights".w1[55] * v2[23] + "NeuroPLC_Weights".w1[56] * v2[24] + "NeuroPLC_Weights".w1[57] * v2[25] + "NeuroPLC_Weights".w1[58] * v2[26] + "NeuroPLC_Weights".w1[59] * v2[27] + "NeuroPLC_Weights".w1[60] * v2[28] + "NeuroPLC_Weights".w1[61] * v2[29] + "NeuroPLC_Weights".w1[62] * v2[30] + "NeuroPLC_Weights".w1[63] * v2[31];
    v3[2] := "NeuroPLC_Weights".w1[512 + 2] + "NeuroPLC_Weights".w1[64] * v2[0] + "NeuroPLC_Weights".w1[65] * v2[1] + "NeuroPLC_Weights".w1[66] * v2[2] + "NeuroPLC_Weights".w1[67] * v2[3] + "NeuroPLC_Weights".w1[68] * v2[4] + "NeuroPLC_Weights".w1[69] * v2[5] + "NeuroPLC_Weights".w1[70] * v2[6] + "NeuroPLC_Weights".w1[71] * v2[7] + "NeuroPLC_Weights".w1[72] * v2[8] + "NeuroPLC_Weights".w1[73] * v2[9] + "NeuroPLC_Weights".w1[74] * v2[10] + "NeuroPLC_Weights".w1[75] * v2[11] + "NeuroPLC_Weights".w1[76] * v2[12] + "NeuroPLC_Weights".w1[77] * v2[13] + "NeuroPLC_Weights".w1[78] * v2[14] + "NeuroPLC_Weights".w1[79] * v2[15] + "NeuroPLC_Weights".w1[80] * v2[16] + "NeuroPLC_Weights".w1[81] * v2[17] + "NeuroPLC_Weights".w1[82] * v2[18] + "NeuroPLC_Weights".w1[83] * v2[19] + "NeuroPLC_Weights".w1[84] * v2[20] + "NeuroPLC_Weights".w1[85] * v2[21] + "NeuroPLC_Weights".w1[86] * v2[22] + "NeuroPLC_Weights".w1[87] * v2[23] + "NeuroPLC_Weights".w1[88] * v2[24] + "NeuroPLC_Weights".w1[89] * v2[25] + "NeuroPLC_Weights".w1[90] * v2[26] + "NeuroPLC_Weights".w1[91] * v2[27] + "NeuroPLC_Weights".w1[92] * v2[28] + "NeuroPLC_Weights".w1[93] * v2[29] + "NeuroPLC_Weights".w1[94] * v2[30] + "NeuroPLC_Weights".w1[95] * v2[31];
    v3[3] := "NeuroPLC_Weights".w1[512 + 3] + "NeuroPLC_Weights".w1[96] * v2[0] + "NeuroPLC_Weights".w1[97] * v2[1] + "NeuroPLC_Weights".w1[98] * v2[2] + "NeuroPLC_Weights".w1[99] * v2[3] + "NeuroPLC_Weights".w1[100] * v2[4] + "NeuroPLC_Weights".w1[101] * v2[5] + "NeuroPLC_Weights".w1[102] * v2[6] + "NeuroPLC_Weights".w1[103] * v2[7] + "NeuroPLC_Weights".w1[104] * v2[8] + "NeuroPLC_Weights".w1[105] * v2[9] + "NeuroPLC_Weights".w1[106] * v2[10] + "NeuroPLC_Weights".w1[107] * v2[11] + "NeuroPLC_Weights".w1[108] * v2[12] + "NeuroPLC_Weights".w1[109] * v2[13] + "NeuroPLC_Weights".w1[110] * v2[14] + "NeuroPLC_Weights".w1[111] * v2[15] + "NeuroPLC_Weights".w1[112] * v2[16] + "NeuroPLC_Weights".w1[113] * v2[17] + "NeuroPLC_Weights".w1[114] * v2[18] + "NeuroPLC_Weights".w1[115] * v2[19] + "NeuroPLC_Weights".w1[116] * v2[20] + "NeuroPLC_Weights".w1[117] * v2[21] + "NeuroPLC_Weights".w1[118] * v2[22] + "NeuroPLC_Weights".w1[119] * v2[23] + "NeuroPLC_Weights".w1[120] * v2[24] + "NeuroPLC_Weights".w1[121] * v2[25] + "NeuroPLC_Weights".w1[122] * v2[26] + "NeuroPLC_Weights".w1[123] * v2[27] + "NeuroPLC_Weights".w1[124] * v2[28] + "NeuroPLC_Weights".w1[125] * v2[29] + "NeuroPLC_Weights".w1[126] * v2[30] + "NeuroPLC_Weights".w1[127] * v2[31];
    v3[4] := "NeuroPLC_Weights".w1[512 + 4] + "NeuroPLC_Weights".w1[128] * v2[0] + "NeuroPLC_Weights".w1[129] * v2[1] + "NeuroPLC_Weights".w1[130] * v2[2] + "NeuroPLC_Weights".w1[131] * v2[3] + "NeuroPLC_Weights".w1[132] * v2[4] + "NeuroPLC_Weights".w1[133] * v2[5] + "NeuroPLC_Weights".w1[134] * v2[6] + "NeuroPLC_Weights".w1[135] * v2[7] + "NeuroPLC_Weights".w1[136] * v2[8] + "NeuroPLC_Weights".w1[137] * v2[9] + "NeuroPLC_Weights".w1[138] * v2[10] + "NeuroPLC_Weights".w1[139] * v2[11] + "NeuroPLC_Weights".w1[140] * v2[12] + "NeuroPLC_Weights".w1[141] * v2[13] + "NeuroPLC_Weights".w1[142] * v2[14] + "NeuroPLC_Weights".w1[143] * v2[15] + "NeuroPLC_Weights".w1[144] * v2[16] + "NeuroPLC_Weights".w1[145] * v2[17] + "NeuroPLC_Weights".w1[146] * v2[18] + "NeuroPLC_Weights".w1[147] * v2[19] + "NeuroPLC_Weights".w1[148] * v2[20] + "NeuroPLC_Weights".w1[149] * v2[21] + "NeuroPLC_Weights".w1[150] * v2[22] + "NeuroPLC_Weights".w1[151] * v2[23] + "NeuroPLC_Weights".w1[152] * v2[24] + "NeuroPLC_Weights".w1[153] * v2[25] + "NeuroPLC_Weights".w1[154] * v2[26] + "NeuroPLC_Weights".w1[155] * v2[27] + "NeuroPLC_Weights".w1[156] * v2[28] + "NeuroPLC_Weights".w1[157] * v2[29] + "NeuroPLC_Weights".w1[158] * v2[30] + "NeuroPLC_Weights".w1[159] * v2[31];
    v3[5] := "NeuroPLC_Weights".w1[512 + 5] + "NeuroPLC_Weights".w1[160] * v2[0] + "NeuroPLC_Weights".w1[161] * v2[1] + "NeuroPLC_Weights".w1[162] * v2[2] + "NeuroPLC_Weights".w1[163] * v2[3] + "NeuroPLC_Weights".w1[164] * v2[4] + "NeuroPLC_Weights".w1[165] * v2[5] + "NeuroPLC_Weights".w1[166] * v2[6] + "NeuroPLC_Weights".w1[167] * v2[7] + "NeuroPLC_Weights".w1[168] * v2[8] + "NeuroPLC_Weights".w1[169] * v2[9] + "NeuroPLC_Weights".w1[170] * v2[10] + "NeuroPLC_Weights".w1[171] * v2[11] + "NeuroPLC_Weights".w1[172] * v2[12] + "NeuroPLC_Weights".w1[173] * v2[13] + "NeuroPLC_Weights".w1[174] * v2[14] + "NeuroPLC_Weights".w1[175] * v2[15] + "NeuroPLC_Weights".w1[176] * v2[16] + "NeuroPLC_Weights".w1[177] * v2[17] + "NeuroPLC_Weights".w1[178] * v2[18] + "NeuroPLC_Weights".w1[179] * v2[19] + "NeuroPLC_Weights".w1[180] * v2[20] + "NeuroPLC_Weights".w1[181] * v2[21] + "NeuroPLC_Weights".w1[182] * v2[22] + "NeuroPLC_Weights".w1[183] * v2[23] + "NeuroPLC_Weights".w1[184] * v2[24] + "NeuroPLC_Weights".w1[185] * v2[25] + "NeuroPLC_Weights".w1[186] * v2[26] + "NeuroPLC_Weights".w1[187] * v2[27] + "NeuroPLC_Weights".w1[188] * v2[28] + "NeuroPLC_Weights".w1[189] * v2[29] + "NeuroPLC_Weights".w1[190] * v2[30] + "NeuroPLC_Weights".w1[191] * v2[31];
    v3[6] := "NeuroPLC_Weights".w1[512 + 6] + "NeuroPLC_Weights".w1[192] * v2[0] + "NeuroPLC_Weights".w1[193] * v2[1] + "NeuroPLC_Weights".w1[194] * v2[2] + "NeuroPLC_Weights".w1[195] * v2[3] + "NeuroPLC_Weights".w1[196] * v2[4] + "NeuroPLC_Weights".w1[197] * v2[5] + "NeuroPLC_Weights".w1[198] * v2[6] + "NeuroPLC_Weights".w1[199] * v2[7] + "NeuroPLC_Weights".w1[200] * v2[8] + "NeuroPLC_Weights".w1[201] * v2[9] + "NeuroPLC_Weights".w1[202] * v2[10] + "NeuroPLC_Weights".w1[203] * v2[11] + "NeuroPLC_Weights".w1[204] * v2[12] + "NeuroPLC_Weights".w1[205] * v2[13] + "NeuroPLC_Weights".w1[206] * v2[14] + "NeuroPLC_Weights".w1[207] * v2[15] + "NeuroPLC_Weights".w1[208] * v2[16] + "NeuroPLC_Weights".w1[209] * v2[17] + "NeuroPLC_Weights".w1[210] * v2[18] + "NeuroPLC_Weights".w1[211] * v2[19] + "NeuroPLC_Weights".w1[212] * v2[20] + "NeuroPLC_Weights".w1[213] * v2[21] + "NeuroPLC_Weights".w1[214] * v2[22] + "NeuroPLC_Weights".w1[215] * v2[23] + "NeuroPLC_Weights".w1[216] * v2[24] + "NeuroPLC_Weights".w1[217] * v2[25] + "NeuroPLC_Weights".w1[218] * v2[26] + "NeuroPLC_Weights".w1[219] * v2[27] + "NeuroPLC_Weights".w1[220] * v2[28] + "NeuroPLC_Weights".w1[221] * v2[29] + "NeuroPLC_Weights".w1[222] * v2[30] + "NeuroPLC_Weights".w1[223] * v2[31];
    v3[7] := "NeuroPLC_Weights".w1[512 + 7] + "NeuroPLC_Weights".w1[224] * v2[0] + "NeuroPLC_Weights".w1[225] * v2[1] + "NeuroPLC_Weights".w1[226] * v2[2] + "NeuroPLC_Weights".w1[227] * v2[3] + "NeuroPLC_Weights".w1[228] * v2[4] + "NeuroPLC_Weights".w1[229] * v2[5] + "NeuroPLC_Weights".w1[230] * v2[6] + "NeuroPLC_Weights".w1[231] * v2[7] + "NeuroPLC_Weights".w1[232] * v2[8] + "NeuroPLC_Weights".w1[233] * v2[9] + "NeuroPLC_Weights".w1[234] * v2[10] + "NeuroPLC_Weights".w1[235] * v2[11] + "NeuroPLC_Weights".w1[236] * v2[12] + "NeuroPLC_Weights".w1[237] * v2[13] + "NeuroPLC_Weights".w1[238] * v2[14] + "NeuroPLC_Weights".w1[239] * v2[15] + "NeuroPLC_Weights".w1[240] * v2[16] + "NeuroPLC_Weights".w1[241] * v2[17] + "NeuroPLC_Weights".w1[242] * v2[18] + "NeuroPLC_Weights".w1[243] * v2[19] + "NeuroPLC_Weights".w1[244] * v2[20] + "NeuroPLC_Weights".w1[245] * v2[21] + "NeuroPLC_Weights".w1[246] * v2[22] + "NeuroPLC_Weights".w1[247] * v2[23] + "NeuroPLC_Weights".w1[248] * v2[24] + "NeuroPLC_Weights".w1[249] * v2[25] + "NeuroPLC_Weights".w1[250] * v2[26] + "NeuroPLC_Weights".w1[251] * v2[27] + "NeuroPLC_Weights".w1[252] * v2[28] + "NeuroPLC_Weights".w1[253] * v2[29] + "NeuroPLC_Weights".w1[254] * v2[30] + "NeuroPLC_Weights".w1[255] * v2[31];
    v3[8] := "NeuroPLC_Weights".w1[512 + 8] + "NeuroPLC_Weights".w1[256] * v2[0] + "NeuroPLC_Weights".w1[257] * v2[1] + "NeuroPLC_Weights".w1[258] * v2[2] + "NeuroPLC_Weights".w1[259] * v2[3] + "NeuroPLC_Weights".w1[260] * v2[4] + "NeuroPLC_Weights".w1[261] * v2[5] + "NeuroPLC_Weights".w1[262] * v2[6] + "NeuroPLC_Weights".w1[263] * v2[7] + "NeuroPLC_Weights".w1[264] * v2[8] + "NeuroPLC_Weights".w1[265] * v2[9] + "NeuroPLC_Weights".w1[266] * v2[10] + "NeuroPLC_Weights".w1[267] * v2[11] + "NeuroPLC_Weights".w1[268] * v2[12] + "NeuroPLC_Weights".w1[269] * v2[13] + "NeuroPLC_Weights".w1[270] * v2[14] + "NeuroPLC_Weights".w1[271] * v2[15] + "NeuroPLC_Weights".w1[272] * v2[16] + "NeuroPLC_Weights".w1[273] * v2[17] + "NeuroPLC_Weights".w1[274] * v2[18] + "NeuroPLC_Weights".w1[275] * v2[19] + "NeuroPLC_Weights".w1[276] * v2[20] + "NeuroPLC_Weights".w1[277] * v2[21] + "NeuroPLC_Weights".w1[278] * v2[22] + "NeuroPLC_Weights".w1[279] * v2[23] + "NeuroPLC_Weights".w1[280] * v2[24] + "NeuroPLC_Weights".w1[281] * v2[25] + "NeuroPLC_Weights".w1[282] * v2[26] + "NeuroPLC_Weights".w1[283] * v2[27] + "NeuroPLC_Weights".w1[284] * v2[28] + "NeuroPLC_Weights".w1[285] * v2[29] + "NeuroPLC_Weights".w1[286] * v2[30] + "NeuroPLC_Weights".w1[287] * v2[31];
    v3[9] := "NeuroPLC_Weights".w1[512 + 9] + "NeuroPLC_Weights".w1[288] * v2[0] + "NeuroPLC_Weights".w1[289] * v2[1] + "NeuroPLC_Weights".w1[290] * v2[2] + "NeuroPLC_Weights".w1[291] * v2[3] + "NeuroPLC_Weights".w1[292] * v2[4] + "NeuroPLC_Weights".w1[293] * v2[5] + "NeuroPLC_Weights".w1[294] * v2[6] + "NeuroPLC_Weights".w1[295] * v2[7] + "NeuroPLC_Weights".w1[296] * v2[8] + "NeuroPLC_Weights".w1[297] * v2[9] + "NeuroPLC_Weights".w1[298] * v2[10] + "NeuroPLC_Weights".w1[299] * v2[11] + "NeuroPLC_Weights".w1[300] * v2[12] + "NeuroPLC_Weights".w1[301] * v2[13] + "NeuroPLC_Weights".w1[302] * v2[14] + "NeuroPLC_Weights".w1[303] * v2[15] + "NeuroPLC_Weights".w1[304] * v2[16] + "NeuroPLC_Weights".w1[305] * v2[17] + "NeuroPLC_Weights".w1[306] * v2[18] + "NeuroPLC_Weights".w1[307] * v2[19] + "NeuroPLC_Weights".w1[308] * v2[20] + "NeuroPLC_Weights".w1[309] * v2[21] + "NeuroPLC_Weights".w1[310] * v2[22] + "NeuroPLC_Weights".w1[311] * v2[23] + "NeuroPLC_Weights".w1[312] * v2[24] + "NeuroPLC_Weights".w1[313] * v2[25] + "NeuroPLC_Weights".w1[314] * v2[26] + "NeuroPLC_Weights".w1[315] * v2[27] + "NeuroPLC_Weights".w1[316] * v2[28] + "NeuroPLC_Weights".w1[317] * v2[29] + "NeuroPLC_Weights".w1[318] * v2[30] + "NeuroPLC_Weights".w1[319] * v2[31];
    v3[10] := "NeuroPLC_Weights".w1[512 + 10] + "NeuroPLC_Weights".w1[320] * v2[0] + "NeuroPLC_Weights".w1[321] * v2[1] + "NeuroPLC_Weights".w1[322] * v2[2] + "NeuroPLC_Weights".w1[323] * v2[3] + "NeuroPLC_Weights".w1[324] * v2[4] + "NeuroPLC_Weights".w1[325] * v2[5] + "NeuroPLC_Weights".w1[326] * v2[6] + "NeuroPLC_Weights".w1[327] * v2[7] + "NeuroPLC_Weights".w1[328] * v2[8] + "NeuroPLC_Weights".w1[329] * v2[9] + "NeuroPLC_Weights".w1[330] * v2[10] + "NeuroPLC_Weights".w1[331] * v2[11] + "NeuroPLC_Weights".w1[332] * v2[12] + "NeuroPLC_Weights".w1[333] * v2[13] + "NeuroPLC_Weights".w1[334] * v2[14] + "NeuroPLC_Weights".w1[335] * v2[15] + "NeuroPLC_Weights".w1[336] * v2[16] + "NeuroPLC_Weights".w1[337] * v2[17] + "NeuroPLC_Weights".w1[338] * v2[18] + "NeuroPLC_Weights".w1[339] * v2[19] + "NeuroPLC_Weights".w1[340] * v2[20] + "NeuroPLC_Weights".w1[341] * v2[21] + "NeuroPLC_Weights".w1[342] * v2[22] + "NeuroPLC_Weights".w1[343] * v2[23] + "NeuroPLC_Weights".w1[344] * v2[24] + "NeuroPLC_Weights".w1[345] * v2[25] + "NeuroPLC_Weights".w1[346] * v2[26] + "NeuroPLC_Weights".w1[347] * v2[27] + "NeuroPLC_Weights".w1[348] * v2[28] + "NeuroPLC_Weights".w1[349] * v2[29] + "NeuroPLC_Weights".w1[350] * v2[30] + "NeuroPLC_Weights".w1[351] * v2[31];
    v3[11] := "NeuroPLC_Weights".w1[512 + 11] + "NeuroPLC_Weights".w1[352] * v2[0] + "NeuroPLC_Weights".w1[353] * v2[1] + "NeuroPLC_Weights".w1[354] * v2[2] + "NeuroPLC_Weights".w1[355] * v2[3] + "NeuroPLC_Weights".w1[356] * v2[4] + "NeuroPLC_Weights".w1[357] * v2[5] + "NeuroPLC_Weights".w1[358] * v2[6] + "NeuroPLC_Weights".w1[359] * v2[7] + "NeuroPLC_Weights".w1[360] * v2[8] + "NeuroPLC_Weights".w1[361] * v2[9] + "NeuroPLC_Weights".w1[362] * v2[10] + "NeuroPLC_Weights".w1[363] * v2[11] + "NeuroPLC_Weights".w1[364] * v2[12] + "NeuroPLC_Weights".w1[365] * v2[13] + "NeuroPLC_Weights".w1[366] * v2[14] + "NeuroPLC_Weights".w1[367] * v2[15] + "NeuroPLC_Weights".w1[368] * v2[16] + "NeuroPLC_Weights".w1[369] * v2[17] + "NeuroPLC_Weights".w1[370] * v2[18] + "NeuroPLC_Weights".w1[371] * v2[19] + "NeuroPLC_Weights".w1[372] * v2[20] + "NeuroPLC_Weights".w1[373] * v2[21] + "NeuroPLC_Weights".w1[374] * v2[22] + "NeuroPLC_Weights".w1[375] * v2[23] + "NeuroPLC_Weights".w1[376] * v2[24] + "NeuroPLC_Weights".w1[377] * v2[25] + "NeuroPLC_Weights".w1[378] * v2[26] + "NeuroPLC_Weights".w1[379] * v2[27] + "NeuroPLC_Weights".w1[380] * v2[28] + "NeuroPLC_Weights".w1[381] * v2[29] + "NeuroPLC_Weights".w1[382] * v2[30] + "NeuroPLC_Weights".w1[383] * v2[31];
    v3[12] := "NeuroPLC_Weights".w1[512 + 12] + "NeuroPLC_Weights".w1[384] * v2[0] + "NeuroPLC_Weights".w1[385] * v2[1] + "NeuroPLC_Weights".w1[386] * v2[2] + "NeuroPLC_Weights".w1[387] * v2[3] + "NeuroPLC_Weights".w1[388] * v2[4] + "NeuroPLC_Weights".w1[389] * v2[5] + "NeuroPLC_Weights".w1[390] * v2[6] + "NeuroPLC_Weights".w1[391] * v2[7] + "NeuroPLC_Weights".w1[392] * v2[8] + "NeuroPLC_Weights".w1[393] * v2[9] + "NeuroPLC_Weights".w1[394] * v2[10] + "NeuroPLC_Weights".w1[395] * v2[11] + "NeuroPLC_Weights".w1[396] * v2[12] + "NeuroPLC_Weights".w1[397] * v2[13] + "NeuroPLC_Weights".w1[398] * v2[14] + "NeuroPLC_Weights".w1[399] * v2[15] + "NeuroPLC_Weights".w1[400] * v2[16] + "NeuroPLC_Weights".w1[401] * v2[17] + "NeuroPLC_Weights".w1[402] * v2[18] + "NeuroPLC_Weights".w1[403] * v2[19] + "NeuroPLC_Weights".w1[404] * v2[20] + "NeuroPLC_Weights".w1[405] * v2[21] + "NeuroPLC_Weights".w1[406] * v2[22] + "NeuroPLC_Weights".w1[407] * v2[23] + "NeuroPLC_Weights".w1[408] * v2[24] + "NeuroPLC_Weights".w1[409] * v2[25] + "NeuroPLC_Weights".w1[410] * v2[26] + "NeuroPLC_Weights".w1[411] * v2[27] + "NeuroPLC_Weights".w1[412] * v2[28] + "NeuroPLC_Weights".w1[413] * v2[29] + "NeuroPLC_Weights".w1[414] * v2[30] + "NeuroPLC_Weights".w1[415] * v2[31];
    v3[13] := "NeuroPLC_Weights".w1[512 + 13] + "NeuroPLC_Weights".w1[416] * v2[0] + "NeuroPLC_Weights".w1[417] * v2[1] + "NeuroPLC_Weights".w1[418] * v2[2] + "NeuroPLC_Weights".w1[419] * v2[3] + "NeuroPLC_Weights".w1[420] * v2[4] + "NeuroPLC_Weights".w1[421] * v2[5] + "NeuroPLC_Weights".w1[422] * v2[6] + "NeuroPLC_Weights".w1[423] * v2[7] + "NeuroPLC_Weights".w1[424] * v2[8] + "NeuroPLC_Weights".w1[425] * v2[9] + "NeuroPLC_Weights".w1[426] * v2[10] + "NeuroPLC_Weights".w1[427] * v2[11] + "NeuroPLC_Weights".w1[428] * v2[12] + "NeuroPLC_Weights".w1[429] * v2[13] + "NeuroPLC_Weights".w1[430] * v2[14] + "NeuroPLC_Weights".w1[431] * v2[15] + "NeuroPLC_Weights".w1[432] * v2[16] + "NeuroPLC_Weights".w1[433] * v2[17] + "NeuroPLC_Weights".w1[434] * v2[18] + "NeuroPLC_Weights".w1[435] * v2[19] + "NeuroPLC_Weights".w1[436] * v2[20] + "NeuroPLC_Weights".w1[437] * v2[21] + "NeuroPLC_Weights".w1[438] * v2[22] + "NeuroPLC_Weights".w1[439] * v2[23] + "NeuroPLC_Weights".w1[440] * v2[24] + "NeuroPLC_Weights".w1[441] * v2[25] + "NeuroPLC_Weights".w1[442] * v2[26] + "NeuroPLC_Weights".w1[443] * v2[27] + "NeuroPLC_Weights".w1[444] * v2[28] + "NeuroPLC_Weights".w1[445] * v2[29] + "NeuroPLC_Weights".w1[446] * v2[30] + "NeuroPLC_Weights".w1[447] * v2[31];
    v3[14] := "NeuroPLC_Weights".w1[512 + 14] + "NeuroPLC_Weights".w1[448] * v2[0] + "NeuroPLC_Weights".w1[449] * v2[1] + "NeuroPLC_Weights".w1[450] * v2[2] + "NeuroPLC_Weights".w1[451] * v2[3] + "NeuroPLC_Weights".w1[452] * v2[4] + "NeuroPLC_Weights".w1[453] * v2[5] + "NeuroPLC_Weights".w1[454] * v2[6] + "NeuroPLC_Weights".w1[455] * v2[7] + "NeuroPLC_Weights".w1[456] * v2[8] + "NeuroPLC_Weights".w1[457] * v2[9] + "NeuroPLC_Weights".w1[458] * v2[10] + "NeuroPLC_Weights".w1[459] * v2[11] + "NeuroPLC_Weights".w1[460] * v2[12] + "NeuroPLC_Weights".w1[461] * v2[13] + "NeuroPLC_Weights".w1[462] * v2[14] + "NeuroPLC_Weights".w1[463] * v2[15] + "NeuroPLC_Weights".w1[464] * v2[16] + "NeuroPLC_Weights".w1[465] * v2[17] + "NeuroPLC_Weights".w1[466] * v2[18] + "NeuroPLC_Weights".w1[467] * v2[19] + "NeuroPLC_Weights".w1[468] * v2[20] + "NeuroPLC_Weights".w1[469] * v2[21] + "NeuroPLC_Weights".w1[470] * v2[22] + "NeuroPLC_Weights".w1[471] * v2[23] + "NeuroPLC_Weights".w1[472] * v2[24] + "NeuroPLC_Weights".w1[473] * v2[25] + "NeuroPLC_Weights".w1[474] * v2[26] + "NeuroPLC_Weights".w1[475] * v2[27] + "NeuroPLC_Weights".w1[476] * v2[28] + "NeuroPLC_Weights".w1[477] * v2[29] + "NeuroPLC_Weights".w1[478] * v2[30] + "NeuroPLC_Weights".w1[479] * v2[31];
    v3[15] := "NeuroPLC_Weights".w1[512 + 15] + "NeuroPLC_Weights".w1[480] * v2[0] + "NeuroPLC_Weights".w1[481] * v2[1] + "NeuroPLC_Weights".w1[482] * v2[2] + "NeuroPLC_Weights".w1[483] * v2[3] + "NeuroPLC_Weights".w1[484] * v2[4] + "NeuroPLC_Weights".w1[485] * v2[5] + "NeuroPLC_Weights".w1[486] * v2[6] + "NeuroPLC_Weights".w1[487] * v2[7] + "NeuroPLC_Weights".w1[488] * v2[8] + "NeuroPLC_Weights".w1[489] * v2[9] + "NeuroPLC_Weights".w1[490] * v2[10] + "NeuroPLC_Weights".w1[491] * v2[11] + "NeuroPLC_Weights".w1[492] * v2[12] + "NeuroPLC_Weights".w1[493] * v2[13] + "NeuroPLC_Weights".w1[494] * v2[14] + "NeuroPLC_Weights".w1[495] * v2[15] + "NeuroPLC_Weights".w1[496] * v2[16] + "NeuroPLC_Weights".w1[497] * v2[17] + "NeuroPLC_Weights".w1[498] * v2[18] + "NeuroPLC_Weights".w1[499] * v2[19] + "NeuroPLC_Weights".w1[500] * v2[20] + "NeuroPLC_Weights".w1[501] * v2[21] + "NeuroPLC_Weights".w1[502] * v2[22] + "NeuroPLC_Weights".w1[503] * v2[23] + "NeuroPLC_Weights".w1[504] * v2[24] + "NeuroPLC_Weights".w1[505] * v2[25] + "NeuroPLC_Weights".w1[506] * v2[26] + "NeuroPLC_Weights".w1[507] * v2[27] + "NeuroPLC_Weights".w1[508] * v2[28] + "NeuroPLC_Weights".w1[509] * v2[29] + "NeuroPLC_Weights".w1[510] * v2[30] + "NeuroPLC_Weights".w1[511] * v2[31];

    // ---- relu1: RELU ----
    IF v3[0] > 0.0 THEN v4[0] := v3[0]; ELSE v4[0] := 0.0; END_IF;
    IF v3[1] > 0.0 THEN v4[1] := v3[1]; ELSE v4[1] := 0.0; END_IF;
    IF v3[2] > 0.0 THEN v4[2] := v3[2]; ELSE v4[2] := 0.0; END_IF;
    IF v3[3] > 0.0 THEN v4[3] := v3[3]; ELSE v4[3] := 0.0; END_IF;
    IF v3[4] > 0.0 THEN v4[4] := v3[4]; ELSE v4[4] := 0.0; END_IF;
    IF v3[5] > 0.0 THEN v4[5] := v3[5]; ELSE v4[5] := 0.0; END_IF;
    IF v3[6] > 0.0 THEN v4[6] := v3[6]; ELSE v4[6] := 0.0; END_IF;
    IF v3[7] > 0.0 THEN v4[7] := v3[7]; ELSE v4[7] := 0.0; END_IF;
    IF v3[8] > 0.0 THEN v4[8] := v3[8]; ELSE v4[8] := 0.0; END_IF;
    IF v3[9] > 0.0 THEN v4[9] := v3[9]; ELSE v4[9] := 0.0; END_IF;
    IF v3[10] > 0.0 THEN v4[10] := v3[10]; ELSE v4[10] := 0.0; END_IF;
    IF v3[11] > 0.0 THEN v4[11] := v3[11]; ELSE v4[11] := 0.0; END_IF;
    IF v3[12] > 0.0 THEN v4[12] := v3[12]; ELSE v4[12] := 0.0; END_IF;
    IF v3[13] > 0.0 THEN v4[13] := v3[13]; ELSE v4[13] := 0.0; END_IF;
    IF v3[14] > 0.0 THEN v4[14] := v3[14]; ELSE v4[14] := 0.0; END_IF;
    IF v3[15] > 0.0 THEN v4[15] := v3[15]; ELSE v4[15] := 0.0; END_IF;

    // ---- fc2: MatMul(16→4) ----
    // W = "NeuroPLC_Weights".w2[:64],   b = w2[64:]
    v5[0] := "NeuroPLC_Weights".w2[64 + 0] + "NeuroPLC_Weights".w2[0] * v4[0] + "NeuroPLC_Weights".w2[1] * v4[1] + "NeuroPLC_Weights".w2[2] * v4[2] + "NeuroPLC_Weights".w2[3] * v4[3] + "NeuroPLC_Weights".w2[4] * v4[4] + "NeuroPLC_Weights".w2[5] * v4[5] + "NeuroPLC_Weights".w2[6] * v4[6] + "NeuroPLC_Weights".w2[7] * v4[7] + "NeuroPLC_Weights".w2[8] * v4[8] + "NeuroPLC_Weights".w2[9] * v4[9] + "NeuroPLC_Weights".w2[10] * v4[10] + "NeuroPLC_Weights".w2[11] * v4[11] + "NeuroPLC_Weights".w2[12] * v4[12] + "NeuroPLC_Weights".w2[13] * v4[13] + "NeuroPLC_Weights".w2[14] * v4[14] + "NeuroPLC_Weights".w2[15] * v4[15];
    v5[1] := "NeuroPLC_Weights".w2[64 + 1] + "NeuroPLC_Weights".w2[16] * v4[0] + "NeuroPLC_Weights".w2[17] * v4[1] + "NeuroPLC_Weights".w2[18] * v4[2] + "NeuroPLC_Weights".w2[19] * v4[3] + "NeuroPLC_Weights".w2[20] * v4[4] + "NeuroPLC_Weights".w2[21] * v4[5] + "NeuroPLC_Weights".w2[22] * v4[6] + "NeuroPLC_Weights".w2[23] * v4[7] + "NeuroPLC_Weights".w2[24] * v4[8] + "NeuroPLC_Weights".w2[25] * v4[9] + "NeuroPLC_Weights".w2[26] * v4[10] + "NeuroPLC_Weights".w2[27] * v4[11] + "NeuroPLC_Weights".w2[28] * v4[12] + "NeuroPLC_Weights".w2[29] * v4[13] + "NeuroPLC_Weights".w2[30] * v4[14] + "NeuroPLC_Weights".w2[31] * v4[15];
    v5[2] := "NeuroPLC_Weights".w2[64 + 2] + "NeuroPLC_Weights".w2[32] * v4[0] + "NeuroPLC_Weights".w2[33] * v4[1] + "NeuroPLC_Weights".w2[34] * v4[2] + "NeuroPLC_Weights".w2[35] * v4[3] + "NeuroPLC_Weights".w2[36] * v4[4] + "NeuroPLC_Weights".w2[37] * v4[5] + "NeuroPLC_Weights".w2[38] * v4[6] + "NeuroPLC_Weights".w2[39] * v4[7] + "NeuroPLC_Weights".w2[40] * v4[8] + "NeuroPLC_Weights".w2[41] * v4[9] + "NeuroPLC_Weights".w2[42] * v4[10] + "NeuroPLC_Weights".w2[43] * v4[11] + "NeuroPLC_Weights".w2[44] * v4[12] + "NeuroPLC_Weights".w2[45] * v4[13] + "NeuroPLC_Weights".w2[46] * v4[14] + "NeuroPLC_Weights".w2[47] * v4[15];
    v5[3] := "NeuroPLC_Weights".w2[64 + 3] + "NeuroPLC_Weights".w2[48] * v4[0] + "NeuroPLC_Weights".w2[49] * v4[1] + "NeuroPLC_Weights".w2[50] * v4[2] + "NeuroPLC_Weights".w2[51] * v4[3] + "NeuroPLC_Weights".w2[52] * v4[4] + "NeuroPLC_Weights".w2[53] * v4[5] + "NeuroPLC_Weights".w2[54] * v4[6] + "NeuroPLC_Weights".w2[55] * v4[7] + "NeuroPLC_Weights".w2[56] * v4[8] + "NeuroPLC_Weights".w2[57] * v4[9] + "NeuroPLC_Weights".w2[58] * v4[10] + "NeuroPLC_Weights".w2[59] * v4[11] + "NeuroPLC_Weights".w2[60] * v4[12] + "NeuroPLC_Weights".w2[61] * v4[13] + "NeuroPLC_Weights".w2[62] * v4[14] + "NeuroPLC_Weights".w2[63] * v4[15];

    // ---- softmax: Softmax ----
    softmax_out[0] := EXP(v5[0]);
    softmax_out[1] := EXP(v5[1]);
    softmax_out[2] := EXP(v5[2]);
    softmax_out[3] := EXP(v5[3]);
    sum_val := softmax_out[0]
             + softmax_out[1]
             + softmax_out[2]
             + softmax_out[3]
             ;
    IF sum_val > 0.0 THEN
        softmax_out[0] := softmax_out[0] / sum_val;
        softmax_out[1] := softmax_out[1] / sum_val;
        softmax_out[2] := softmax_out[2] / sum_val;
        softmax_out[3] := softmax_out[3] / sum_val;
    END_IF;

    // ---- Argmax ----
    max_val := softmax_out[0];
    fault_class := 0;
    IF softmax_out[1] > max_val THEN
        max_val := softmax_out[1];
        fault_class := 1;
    END_IF;
    IF softmax_out[2] > max_val THEN
        max_val := softmax_out[2];
        fault_class := 2;
    END_IF;
    IF softmax_out[3] > max_val THEN
        max_val := softmax_out[3];
        fault_class := 3;
    END_IF;
    confidence := max_val;

END_FUNCTION_BLOCK